LIN {X 0,Y 249.004,Z 223.47,A -85,B 0,C 180,E1 -19037.36,E2 -19037.36} C_VEL
LIN {X 0,Y 249.044,Z 223.457,A -85,B 0,C 180,E1 -19042.201,E2 -19042.201} C_VEL
LIN {X 0,Y 249.045,Z 223.461,A -85,B 0,C 180,E1 -19045.64,E2 -19045.64} C_VEL
LIN {X 0,Y 249.004,Z 223.467,A -85,B 0,C 180,E1 -19049.467,E2 -19049.467} C_VEL
LIN {X 0,Y 249.038,Z 223.46,A -85,B 0,C 180,E1 -19053.158,E2 -19053.158} C_VEL
LIN {X 0,Y 249.057,Z 223.459,A -85,B 0,C 180,E1 -19056.73,E2 -19056.73} C_VEL
LIN {X 0,Y 249.089,Z 223.455,A -85,B 0,C 180,E1 -19060.21,E2 -19060.21} C_VEL
LIN {X 0,Y 249.199,Z 223.439,A -85,B 0,C 180,E1 -19063.619,E2 -19063.619} C_VEL
LIN {X 0,Y 249.237,Z 223.426,A -85,B 0,C 180,E1 -19068.616,E2 -19068.616} C_VEL
LIN {X 0,Y 249.421,Z 223.401,A -85,B 0,C 180,E1 -19071.901,E2 -19071.901} C_VEL
LIN {X 0,Y 249.275,Z 223.429,A -85,B 0,C 180,E1 -19075.148,E2 -19075.148} C_VEL
LIN {X 0,Y 249.67,Z 223.386,A -85,B 0,C 180,E1 -19078.387,E2 -19078.387} C_VEL
LIN {X 0,Y 249.664,Z 223.384,A -85,B 0,C 180,E1 -19081.613,E2 -19081.613} C_VEL
LIN {X 0,Y 249.432,Z 223.406,A -85,B 0,C 180,E1 -19086.471,E2 -19086.471} C_VEL
LIN {X 0,Y 249.346,Z 223.417,A -85,B 0,C 180,E1 -19089.736,E2 -19089.736} C_VEL
LIN {X 0,Y 249.166,Z 223.447,A -85,B 0,C 180,E1 -19094.706,E2 -19094.706} C_VEL
LIN {X 0,Y 249.108,Z 223.454,A -85,B 0,C 180,E1 -19098.12,E2 -19098.12} C_VEL
LIN {X 0,Y 248.362,Z 223.545,A -85,B 0,C 180,E1 -19099.469,E2 -19099.469} C_VEL
LIN {X 0,Y 245.448,Z 223.906,A -85,B 0,C 180,E1 -19101.666,E2 -19101.666} C_VEL
LIN {X 0,Y 243.036,Z 224.209,A -85,B 0,C 180,E1 -19103.456,E2 -19103.456} C_VEL
LIN {X 0,Y 242.037,Z 224.335,A -85,B 0,C 180,E1 -19104.845,E2 -19104.845} C_VEL
LIN {X 0,Y 241.972,Z 224.344,A -85,B 0,C 180,E1 -19105.316,E2 -19105.316} C_VEL
LIN {X 0,Y 241.971,Z 224.343,A -85,B 0,C 180,E1 -19109.588,E2 -19109.588} C_VEL
LIN {X 0,Y 241.982,Z 224.344,A -85,B 0,C 180,E1 -19113.493,E2 -19113.493} C_VEL
LIN {X 0,Y 241.986,Z 224.345,A -85,B 0,C 180,E1 -19117.583,E2 -19117.583} C_VEL
LIN {X 0,Y 241.912,Z 224.352,A -85,B 0,C 180,E1 -19121.928,E2 -19121.928} C_VEL
LIN {X 0,Y 241.903,Z 224.351,A -85,B 0,C 180,E1 -19126.58,E2 -19126.58} C_VEL
LIN {X 0,Y 241.997,Z 224.342,A -85,B 0,C 180,E1 -19131.64,E2 -19131.64} C_VEL
LIN {X 0,Y 242.029,Z 224.408,A -85,B 0,C 180,E1 -19132.328,E2 -19132.328} C_VEL
LIN {X 0,Y 244.612,Z 236.152,A -85,B 0,C 180,E1 -19136.43,E2 -19136.43} C_VEL
LIN {X 0,Y 247.148,Z 248.776,A -85,B 0,C 180,E1 -19140.577,E2 -19140.577} C_VEL
LIN {X 0,Y 249.712,Z 271.884,A -85,B 0,C 180,E1 -19141.664,E2 -19141.664} C_VEL
LIN {X 0,Y 253.2,Z 306.04,A -85,B 0,C 180,E1 -19143.192,E2 -19143.192} C_VEL
LIN {X 0,Y 251.212,Z 359.282,A -85,B 0,C 180,E1 -19145.022,E2 -19145.022} C_VEL
LIN {X 0,Y 250.257,Z 372.001,A -85,B 0,C 180,E1 -19145.75,E2 -19145.75} C_VEL
LIN {X 0,Y 248.888,Z 385.038,A -85,B 0,C 180,E1 -19146.823,E2 -19146.823} C_VEL
LIN {X 0,Y 247.113,Z 398.148,A -85,B 0,C 180,E1 -19148.301,E2 -19148.301} C_VEL
LIN {X 0,Y 245.54,Z 409.14,A -85,B 0,C 180,E1 -19149.911,E2 -19149.911} C_VEL
LIN {X 0,Y 243.962,Z 419.427,A -85,B 0,C 180,E1 -19151.814,E2 -19151.814} C_VEL
LIN {X 0,Y 242.778,Z 427.354,A -85,B 0,C 180,E1 -19153.605,E2 -19153.605} C_VEL
LIN {X 0,Y 241.628,Z 436.389,A -85,B 0,C 180,E1 -19156.115,E2 -19156.115} C_VEL
LIN {X 0,Y 240.728,Z 443.544,A -85,B 0,C 180,E1 -19158.634,E2 -19158.634} C_VEL
LIN {X 0,Y 240.323,Z 450.068,A -85,B 0,C 180,E1 -19161.592,E2 -19161.592} C_VEL
LIN {X 0,Y 240.317,Z 453.94,A -85,B 0,C 180,E1 -19163.892,E2 -19163.892} C_VEL
LIN {X 0,Y 240.292,Z 457.328,A -85,B 0,C 180,E1 -19166.646,E2 -19166.646} C_VEL
LIN {X 0,Y 240.448,Z 458.797,A -85,B 0,C 180,E1 -19168.325,E2 -19168.325} C_VEL
LIN {X 0,Y 240.644,Z 459.779,A -85,B 0,C 180,E1 -19170,E2 -19170} C_VEL
LIN {X 0,Y 240.335,Z 460.292,A -85,B 0,C 180,E1 -19171.675,E2 -19171.675} C_VEL
LIN {X 0,Y 240.15,Z 460.406,A -85,B 0,C 180,E1 -19173.355,E2 -19173.355} C_VEL
LIN {X 0,Y 239.968,Z 460.015,A -85,B 0,C 180,E1 -19175.272,E2 -19175.272} C_VEL
LIN {X 0,Y 240.126,Z 458.23,A -85,B 0,C 180,E1 -19178.414,E2 -19178.414} C_VEL
LIN {X 0,Y 240.395,Z 456.694,A -85,B 0,C 180,E1 -19180.102,E2 -19180.102} C_VEL
LIN {X 0,Y 241.109,Z 453.576,A -85,B 0,C 180,E1 -19182.627,E2 -19182.627} C_VEL
LIN {X 0,Y 242.499,Z 449.461,A -85,B 0,C 180,E1 -19185.119,E2 -19185.119} C_VEL
LIN {X 0,Y 244.576,Z 443.266,A -85,B 0,C 180,E1 -19187.993,E2 -19187.993} C_VEL
LIN {X 0,Y 246.746,Z 436.536,A -85,B 0,C 180,E1 -19190.42,E2 -19190.42} C_VEL
LIN {X 0,Y 249.644,Z 428.244,A -85,B 0,C 180,E1 -19192.773,E2 -19192.773} C_VEL
LIN {X 0,Y 253.105,Z 418.103,A -85,B 0,C 180,E1 -19195.052,E2 -19195.052} C_VEL
LIN {X 0,Y 256.227,Z 407.616,A -85,B 0,C 180,E1 -19196.909,E2 -19196.909} C_VEL
LIN {X 0,Y 259.456,Z 395.965,A -85,B 0,C 180,E1 -19198.516,E2 -19198.516} C_VEL
LIN {X 0,Y 262.177,Z 384.572,A -85,B 0,C 180,E1 -19199.73,E2 -19199.73} C_VEL
LIN {X 0,Y 264.726,Z 371.887,A -85,B 0,C 180,E1 -19200.734,E2 -19200.734} C_VEL
LIN {X 0,Y 266.699,Z 358.144,A -85,B 0,C 180,E1 -19201.528,E2 -19201.528} C_VEL
LIN {X 0,Y 268.166,Z 340.024,A -85,B 0,C 180,E1 -19202.191,E2 -19202.191} C_VEL
LIN {X 0,Y 270.151,Z 309.712,A -85,B 0,C 180,E1 -19203.199,E2 -19203.199} C_VEL
LIN {X 0,Y 268.902,Z 293.084,A -85,B 0,C 180,E1 -19204.25,E2 -19204.25} C_VEL
LIN {X 0,Y 266.92,Z 276.84,A -85,B 0,C 180,E1 -19205.487,E2 -19205.487} C_VEL
LIN {X 0,Y 263.665,Z 268.777,A -85,B 0,C 180,E1 -19206.696,E2 -19206.696} C_VEL
LIN {X 0,Y 259.896,Z 260.954,A -85,B 0,C 180,E1 -19208.095,E2 -19208.095} C_VEL
LIN {X 0,Y 257.167,Z 255.727,A -85,B 0,C 180,E1 -19209.168,E2 -19209.168} C_VEL
LIN {X 0,Y 254.586,Z 251.104,A -85,B 0,C 180,E1 -19210.228,E2 -19210.228} C_VEL
LIN {X 0,Y 250.869,Z 244.957,A -85,B 0,C 180,E1 -19211.84,E2 -19211.84} C_VEL
LIN {X 0,Y 246.986,Z 238.614,A -85,B 0,C 180,E1 -19213.774,E2 -19213.774} C_VEL
LIN {X 0,Y 244.929,Z 232.476,A -85,B 0,C 180,E1 -19217.6,E2 -19217.6} C_VEL
LIN {X 0,Y 243.229,Z 227.568,A -85,B 0,C 180,E1 -19221.274,E2 -19221.274} C_VEL
LIN {X 0,Y 242.005,Z 224.336,A -85,B 0,C 180,E1 -19224.403,E2 -19224.403} C_VEL
LIN {X 0,Y 241.953,Z 224.342,A -85,B 0,C 180,E1 -19228.476,E2 -19228.476} C_VEL
LIN {X 0,Y 241.969,Z 224.343,A -85,B 0,C 180,E1 -19232.308,E2 -19232.308} C_VEL
LIN {X 0,Y 242.026,Z 224.331,A -85,B 0,C 180,E1 -19236.012,E2 -19236.012} C_VEL
LIN {X 0,Y 242.022,Z 224.33,A -85,B 0,C 180,E1 -19239.606,E2 -19239.606} C_VEL
LIN {X 0,Y 242.115,Z 224.321,A -85,B 0,C 180,E1 -19243.316,E2 -19243.316} C_VEL
LIN {X 0,Y 242.154,Z 224.318,A -85,B 0,C 180,E1 -19246.574,E2 -19246.574} C_VEL
LIN {X 0,Y 242.4,Z 224.286,A -85,B 0,C 180,E1 -19251.664,E2 -19251.664} C_VEL
LIN {X 0,Y 242.421,Z 224.433,A -85,B 0,C 180,E1 -19252.451,E2 -19252.451} C_VEL
LIN {X 0,Y 243.17,Z 226.719,A -85,B 0,C 180,E1 -19252.996,E2 -19252.996} C_VEL
LIN {X 0,Y 245.186,Z 229.149,A -85,B 0,C 180,E1 -19254.098,E2 -19254.098} C_VEL
LIN {X 0,Y 246.596,Z 230.283,A -85,B 0,C 180,E1 -19254.789,E2 -19254.789} C_VEL
LIN {X 0,Y 248.318,Z 233.194,A -85,B 0,C 180,E1 -19255.688,E2 -19255.688} C_VEL
LIN {X 0,Y 250.915,Z 235.599,A -85,B 0,C 180,E1 -19256.82,E2 -19256.82} C_VEL
LIN {X 0,Y 253.281,Z 239.028,A -85,B 0,C 180,E1 -19257.877,E2 -19257.877} C_VEL
LIN {X 0,Y 254.718,Z 240.902,A -85,B 0,C 180,E1 -19258.464,E2 -19258.464} C_VEL
LIN {X 0,Y 257.831,Z 245.506,A -85,B 0,C 180,E1 -19259.698,E2 -19259.698} C_VEL
LIN {X 0,Y 265.688,Z 258.053,A -85,B 0,C 180,E1 -19262.526,E2 -19262.526} C_VEL
LIN {X 0,Y 270.454,Z 266.96,A -85,B 0,C 180,E1 -19264.103,E2 -19264.103} C_VEL
LIN {X 0,Y 272.41,Z 270.959,A -85,B 0,C 180,E1 -19264.719,E2 -19264.719} C_VEL
LIN {X 0,Y 268.634,Z 326.119,A -85,B 0,C 180,E1 -19266.582,E2 -19266.582} C_VEL
LIN {X 0,Y 267.326,Z 338.992,A -85,B 0,C 180,E1 -19267.297,E2 -19267.297} C_VEL
LIN {X 0,Y 265.555,Z 351.406,A -85,B 0,C 180,E1 -19268.274,E2 -19268.274} C_VEL
LIN {X 0,Y 263.204,Z 363.778,A -85,B 0,C 180,E1 -19269.568,E2 -19269.568} C_VEL
LIN {X 0,Y 260.667,Z 374.697,A -85,B 0,C 180,E1 -19271.046,E2 -19271.046} C_VEL
LIN {X 0,Y 257.859,Z 384.956,A -85,B 0,C 180,E1 -19272.794,E2 -19272.794} C_VEL
LIN {X 0,Y 254.955,Z 394.175,A -85,B 0,C 180,E1 -19274.783,E2 -19274.783} C_VEL
LIN {X 0,Y 252.106,Z 402.348,A -85,B 0,C 180,E1 -19276.998,E2 -19276.998} C_VEL
LIN {X 0,Y 249.515,Z 409.181,A -85,B 0,C 180,E1 -19279.327,E2 -19279.327} C_VEL
LIN {X 0,Y 247.225,Z 414.655,A -85,B 0,C 180,E1 -19281.688,E2 -19281.688} C_VEL
LIN {X 0,Y 244.992,Z 419.645,A -85,B 0,C 180,E1 -19284.579,E2 -19284.579} C_VEL
LIN {X 0,Y 243.177,Z 423.206,A -85,B 0,C 180,E1 -19287.543,E2 -19287.543} C_VEL
LIN {X 0,Y 242.202,Z 424.804,A -85,B 0,C 180,E1 -19289.557,E2 -19289.557} C_VEL
LIN {X 0,Y 241.18,Z 425.997,A -85,B 0,C 180,E1 -19292.322,E2 -19292.322} C_VEL
LIN {X 0,Y 240.526,Z 426.078,A -85,B 0,C 180,E1 -19295.102,E2 -19295.102} C_VEL
LIN {X 0,Y 240.229,Z 425.025,A -85,B 0,C 180,E1 -19297.906,E2 -19297.906} C_VEL
LIN {X 0,Y 240.205,Z 423.052,A -85,B 0,C 180,E1 -19300.473,E2 -19300.473} C_VEL
LIN {X 0,Y 240.581,Z 419.994,A -85,B 0,C 180,E1 -19303.088,E2 -19303.088} C_VEL
LIN {X 0,Y 241.163,Z 415.077,A -85,B 0,C 180,E1 -19306.098,E2 -19306.098} C_VEL
LIN {X 0,Y 241.859,Z 409.983,A -85,B 0,C 180,E1 -19308.464,E2 -19308.464} C_VEL
LIN {X 0,Y 242.782,Z 403.678,A -85,B 0,C 180,E1 -19310.816,E2 -19310.816} C_VEL
LIN {X 0,Y 244.097,Z 395.086,A -85,B 0,C 180,E1 -19313.375,E2 -19313.375} C_VEL
LIN {X 0,Y 245.483,Z 385.904,A -85,B 0,C 180,E1 -19315.575,E2 -19315.575} C_VEL
LIN {X 0,Y 246.977,Z 375.589,A -85,B 0,C 180,E1 -19317.553,E2 -19317.553} C_VEL
LIN {X 0,Y 248.499,Z 363.511,A -85,B 0,C 180,E1 -19319.398,E2 -19319.398} C_VEL
LIN {X 0,Y 249.898,Z 351.267,A -85,B 0,C 180,E1 -19320.836,E2 -19320.836} C_VEL
LIN {X 0,Y 251.035,Z 338.511,A -85,B 0,C 180,E1 -19321.971,E2 -19321.971} C_VEL
LIN {X 0,Y 251.729,Z 325.929,A -85,B 0,C 180,E1 -19322.781,E2 -19322.781} C_VEL
LIN {X 0,Y 252.39,Z 309.148,A -85,B 0,C 180,E1 -19323.438,E2 -19323.438} C_VEL
LIN {X 0,Y 254.486,Z 255.593,A -85,B 0,C 180,E1 -19325.202,E2 -19325.202} C_VEL
LIN {X 0,Y 244.932,Z 231.694,A -85,B 0,C 180,E1 -19326.909,E2 -19326.909} C_VEL
LIN {X 0,Y 242.099,Z 224.79,A -85,B 0,C 180,E1 -19327.436,E2 -19327.436} C_VEL
LIN {X 0,Y 242.005,Z 224.341,A -85,B 0,C 180,E1 -19327.483,E2 -19327.483} C_VEL
LIN {X 0,Y 242.05,Z 224.334,A -85,B 0,C 180,E1 -19331.375,E2 -19331.375} C_VEL
LIN {X 0,Y 242.14,Z 224.324,A -85,B 0,C 180,E1 -19334.858,E2 -19334.858} C_VEL
LIN {X 0,Y 242.343,Z 224.299,A -85,B 0,C 180,E1 -19340.405,E2 -19340.405} C_VEL
LIN {X 0,Y 242.401,Z 224.289,A -85,B 0,C 180,E1 -19343.341,E2 -19343.341} C_VEL
LIN {X 0,Y 242.634,Z 224.262,A -85,B 0,C 180,E1 -19348.341,E2 -19348.341} C_VEL
LIN {X 0,Y 242.632,Z 224.259,A -85,B 0,C 180,E1 -19351.66,E2 -19351.66} C_VEL
LIN {X 0,Y 242.408,Z 224.289,A -85,B 0,C 180,E1 -19356.66,E2 -19356.66} C_VEL
LIN {X 0,Y 242.269,Z 224.307,A -85,B 0,C 180,E1 -19360.024,E2 -19360.024} C_VEL
LIN {X 0,Y 242.169,Z 224.317,A -85,B 0,C 180,E1 -19365.141,E2 -19365.141} C_VEL
LIN {X 0,Y 242.074,Z 224.327,A -85,B 0,C 180,E1 -19368.625,E2 -19368.625} C_VEL
LIN {X 0,Y 242.007,Z 224.332,A -85,B 0,C 180,E1 -19372.181,E2 -19372.181} C_VEL
LIN {X 0,Y 242.034,Z 224.335,A -85,B 0,C 180,E1 -19375.821,E2 -19375.821} C_VEL
LIN {X 0,Y 241.971,Z 224.345,A -85,B 0,C 180,E1 -19379.589,E2 -19379.589} C_VEL
LIN {X 0,Y 241.981,Z 224.34,A -85,B 0,C 180,E1 -19383.493,E2 -19383.493} C_VEL
LIN {X 0,Y 241.985,Z 224.327,A -85,B 0,C 180,E1 -19387.583,E2 -19387.583} C_VEL
LIN {X 0,Y 241.929,Z 224.344,A -85,B 0,C 180,E1 -19391.925,E2 -19391.925} C_VEL
LIN {X 0,Y 241.922,Z 224.348,A -85,B 0,C 180,E1 -19396.575,E2 -19396.575} C_VEL
LIN {X 0,Y 241.995,Z 224.337,A -85,B 0,C 180,E1 -19401.641,E2 -19401.641} C_VEL
LIN {X 0,Y 241.989,Z 224.336,A -85,B 0,C 180,E1 -19404.489,E2 -19404.489} C_VEL
LIN {X 0,Y 241.955,Z 224.344,A -85,B 0,C 180,E1 -19408.477,E2 -19408.477} C_VEL
LIN {X 0,Y 241.97,Z 224.34,A -85,B 0,C 180,E1 -19412.308,E2 -19412.308} C_VEL
LIN {X 0,Y 242.027,Z 224.331,A -85,B 0,C 180,E1 -19416.013,E2 -19416.013} C_VEL
LIN {X 0,Y 242.024,Z 224.335,A -85,B 0,C 180,E1 -19419.607,E2 -19419.607} C_VEL
LIN {X 0,Y 242.13,Z 224.32,A -85,B 0,C 180,E1 -19423.307,E2 -19423.307} C_VEL
LIN {X 0,Y 242.171,Z 224.308,A -85,B 0,C 180,E1 -19428.279,E2 -19428.279} C_VEL
LIN {X 0,Y 242.375,Z 224.277,A -85,B 0,C 180,E1 -19431.664,E2 -19431.664} C_VEL
LIN {X 0,Y 242.236,Z 224.306,A -85,B 0,C 180,E1 -19435.007,E2 -19435.007} C_VEL
LIN {X 0,Y 242.63,Z 224.262,A -85,B 0,C 180,E1 -19438.34,E2 -19438.34} C_VEL
LIN {X 0,Y 242.623,Z 224.261,A -85,B 0,C 180,E1 -19441.66,E2 -19441.66} C_VEL
LIN {X 0,Y 242.404,Z 224.279,A -85,B 0,C 180,E1 -19446.66,E2 -19446.66} C_VEL
LIN {X 0,Y 242.269,Z 224.3,A -85,B 0,C 180,E1 -19450.024,E2 -19450.024} C_VEL
LIN {X 0,Y 242.129,Z 224.324,A -85,B 0,C 180,E1 -19455.143,E2 -19455.143} C_VEL
LIN {X 0,Y 242.049,Z 224.331,A -85,B 0,C 180,E1 -19458.626,E2 -19458.626} C_VEL
LIN {X 0,Y 241.991,Z 224.339,A -85,B 0,C 180,E1 -19462.182,E2 -19462.182} C_VEL
LIN {X 0,Y 241.972,Z 224.344,A -85,B 0,C 180,E1 -19465.316,E2 -19465.316} C_VEL
LIN {X 0,Y 241.353,Z 224.425,A -85,B 0,C 180,E1 -19466.705,E2 -19466.705} C_VEL
LIN {X 0,Y 238.537,Z 224.775,A -85,B 0,C 180,E1 -19468.972,E2 -19468.972} C_VEL
LIN {X 0,Y 236.106,Z 225.073,A -85,B 0,C 180,E1 -19470.819,E2 -19470.819} C_VEL
LIN {X 0,Y 235.045,Z 225.205,A -85,B 0,C 180,E1 -19472.252,E2 -19472.252} C_VEL
LIN {X 0,Y 234.95,Z 225.216,A -85,B 0,C 180,E1 -19472.738,E2 -19472.738} C_VEL
LIN {X 0,Y 234.918,Z 225.221,A -85,B 0,C 180,E1 -19476.751,E2 -19476.751} C_VEL
LIN {X 0,Y 234.914,Z 225.224,A -85,B 0,C 180,E1 -19478.935,E2 -19478.935} C_VEL
LIN {X 0,Y 234.855,Z 225.233,A -85,B 0,C 180,E1 -19483.494,E2 -19483.494} C_VEL
LIN {X 0,Y 234.856,Z 225.229,A -85,B 0,C 180,E1 -19486.506,E2 -19486.506} C_VEL
LIN {X 0,Y 234.972,Z 225.217,A -85,B 0,C 180,E1 -19491.774,E2 -19491.774} C_VEL
LIN {X 0,Y 236.986,Z 234.459,A -85,B 0,C 180,E1 -19495.188,E2 -19495.188} C_VEL
LIN {X 0,Y 239.364,Z 245.731,A -85,B 0,C 180,E1 -19499.082,E2 -19499.082} C_VEL
LIN {X 0,Y 239.85,Z 248.256,A -85,B 0,C 180,E1 -19499.905,E2 -19499.905} C_VEL
LIN {X 0,Y 241.048,Z 253.117,A -85,B 0,C 180,E1 -19500.204,E2 -19500.204} C_VEL
LIN {X 0,Y 246.464,Z 306.984,A -85,B 0,C 180,E1 -19502.71,E2 -19502.71} C_VEL
LIN {X 0,Y 244.423,Z 358.04,A -85,B 0,C 180,E1 -19504.506,E2 -19504.506} C_VEL
LIN {X 0,Y 243.525,Z 370.993,A -85,B 0,C 180,E1 -19505.262,E2 -19505.262} C_VEL
LIN {X 0,Y 242.077,Z 384.148,A -85,B 0,C 180,E1 -19506.358,E2 -19506.358} C_VEL
LIN {X 0,Y 240.52,Z 395.755,A -85,B 0,C 180,E1 -19507.674,E2 -19507.674} C_VEL
LIN {X 0,Y 238.876,Z 407.102,A -85,B 0,C 180,E1 -19509.325,E2 -19509.325} C_VEL
LIN {X 0,Y 237.422,Z 416.33,A -85,B 0,C 180,E1 -19510.997,E2 -19510.997} C_VEL
LIN {X 0,Y 235.854,Z 425.804,A -85,B 0,C 180,E1 -19513.11,E2 -19513.11} C_VEL
LIN {X 0,Y 234.679,Z 435.015,A -85,B 0,C 180,E1 -19515.696,E2 -19515.696} C_VEL
LIN {X 0,Y 233.729,Z 442.37,A -85,B 0,C 180,E1 -19518.289,E2 -19518.289} C_VEL
LIN {X 0,Y 233.34,Z 447.316,A -85,B 0,C 180,E1 -19520.464,E2 -19520.464} C_VEL
LIN {X 0,Y 233.202,Z 452.07,A -85,B 0,C 180,E1 -19523.076,E2 -19523.076} C_VEL
LIN {X 0,Y 233.272,Z 454.555,A -85,B 0,C 180,E1 -19524.814,E2 -19524.814} C_VEL
LIN {X 0,Y 233.225,Z 456.519,A -85,B 0,C 180,E1 -19526.544,E2 -19526.544} C_VEL
LIN {X 0,Y 233.365,Z 458.051,A -85,B 0,C 180,E1 -19528.274,E2 -19528.274} C_VEL
LIN {X 0,Y 233.587,Z 459.122,A -85,B 0,C 180,E1 -19530,E2 -19530} C_VEL
LIN {X 0,Y 233.249,Z 459.681,A -85,B 0,C 180,E1 -19531.726,E2 -19531.726} C_VEL
LIN {X 0,Y 233.071,Z 459.842,A -85,B 0,C 180,E1 -19533.457,E2 -19533.457} C_VEL
LIN {X 0,Y 232.897,Z 459.588,A -85,B 0,C 180,E1 -19535.237,E2 -19535.237} C_VEL
LIN {X 0,Y 232.899,Z 458.941,A -85,B 0,C 180,E1 -19536.932,E2 -19536.932} C_VEL
LIN {X 0,Y 233.373,Z 456.383,A -85,B 0,C 180,E1 -19540.409,E2 -19540.409} C_VEL
LIN {X 0,Y 234.161,Z 453.382,A -85,B 0,C 180,E1 -19543.008,E2 -19543.008} C_VEL
LIN {X 0,Y 235.638,Z 449.379,A -85,B 0,C 180,E1 -19545.57,E2 -19545.57} C_VEL
LIN {X 0,Y 237.455,Z 444.269,A -85,B 0,C 180,E1 -19548.105,E2 -19548.105} C_VEL
LIN {X 0,Y 239.664,Z 437.95,A -85,B 0,C 180,E1 -19550.603,E2 -19550.603} C_VEL
LIN {X 0,Y 242.605,Z 430.206,A -85,B 0,C 180,E1 -19553.021,E2 -19553.021} C_VEL
LIN {X 0,Y 245.465,Z 422.389,A -85,B 0,C 180,E1 -19554.98,E2 -19554.98} C_VEL
LIN {X 0,Y 248.945,Z 411.937,A -85,B 0,C 180,E1 -19557.079,E2 -19557.079} C_VEL
LIN {X 0,Y 252.189,Z 401.412,A -85,B 0,C 180,E1 -19558.732,E2 -19558.732} C_VEL
LIN {X 0,Y 255.304,Z 389.924,A -85,B 0,C 180,E1 -19560.157,E2 -19560.157} C_VEL
LIN {X 0,Y 258.063,Z 378.066,A -85,B 0,C 180,E1 -19561.274,E2 -19561.274} C_VEL
LIN {X 0,Y 260.595,Z 364.125,A -85,B 0,C 180,E1 -19562.241,E2 -19562.241} C_VEL
LIN {X 0,Y 262.232,Z 350.287,A -85,B 0,C 180,E1 -19562.895,E2 -19562.895} C_VEL
LIN {X 0,Y 265.041,Z 310.297,A -85,B 0,C 180,E1 -19564.251,E2 -19564.251} C_VEL
LIN {X 0,Y 263.895,Z 294.774,A -85,B 0,C 180,E1 -19565.275,E2 -19565.275} C_VEL
LIN {X 0,Y 262.209,Z 279.646,A -85,B 0,C 180,E1 -19566.477,E2 -19566.477} C_VEL
LIN {X 0,Y 257.444,Z 268.533,A -85,B 0,C 180,E1 -19568.335,E2 -19568.335} C_VEL
LIN {X 0,Y 253.621,Z 260.876,A -85,B 0,C 180,E1 -19569.925,E2 -19569.925} C_VEL
LIN {X 0,Y 251.077,Z 256.261,A -85,B 0,C 180,E1 -19571.019,E2 -19571.019} C_VEL
LIN {X 0,Y 247.526,Z 250.181,A -85,B 0,C 180,E1 -19572.681,E2 -19572.681} C_VEL
LIN {X 0,Y 243.577,Z 243.84,A -85,B 0,C 180,E1 -19574.706,E2 -19574.706} C_VEL
LIN {X 0,Y 239.557,Z 237.626,A -85,B 0,C 180,E1 -19577.067,E2 -19577.067} C_VEL
LIN {X 0,Y 239.211,Z 236.801,A -85,B 0,C 180,E1 -19577.488,E2 -19577.488} C_VEL
LIN {X 0,Y 237.935,Z 233.255,A -85,B 0,C 180,E1 -19580.172,E2 -19580.172} C_VEL
LIN {X 0,Y 237.409,Z 231.555,A -85,B 0,C 180,E1 -19581.562,E2 -19581.562} C_VEL
LIN {X 0,Y 235.745,Z 227.774,A -85,B 0,C 180,E1 -19585.498,E2 -19585.498} C_VEL
LIN {X 0,Y 234.888,Z 225.226,A -85,B 0,C 180,E1 -19588.927,E2 -19588.927} C_VEL
LIN {X 0,Y 234.968,Z 225.209,A -85,B 0,C 180,E1 -19593.806,E2 -19593.806} C_VEL
LIN {X 0,Y 234.99,Z 225.208,A -85,B 0,C 180,E1 -19598.968,E2 -19598.968} C_VEL
LIN {X 0,Y 235.056,Z 225.199,A -85,B 0,C 180,E1 -19603.092,E2 -19603.092} C_VEL
LIN {X 0,Y 235.111,Z 225.192,A -85,B 0,C 180,E1 -19607.922,E2 -19607.922} C_VEL
LIN {X 0,Y 235.173,Z 225.364,A -85,B 0,C 180,E1 -19608.471,E2 -19608.471} C_VEL
LIN {X 0,Y 235.883,Z 227.535,A -85,B 0,C 180,E1 -19609.175,E2 -19609.175} C_VEL
LIN {X 0,Y 237.812,Z 229.766,A -85,B 0,C 180,E1 -19610.554,E2 -19610.554} C_VEL
LIN {X 0,Y 239.977,Z 231.128,A -85,B 0,C 180,E1 -19611.844,E2 -19611.844} C_VEL
LIN {X 0,Y 241.504,Z 234.067,A -85,B 0,C 180,E1 -19612.853,E2 -19612.853} C_VEL
LIN {X 0,Y 244.057,Z 236.636,A -85,B 0,C 180,E1 -19614.215,E2 -19614.215} C_VEL
LIN {X 0,Y 246.175,Z 239.881,A -85,B 0,C 180,E1 -19615.353,E2 -19615.353} C_VEL
LIN {X 0,Y 248.301,Z 242.029,A -85,B 0,C 180,E1 -19616.317,E2 -19616.317} C_VEL
LIN {X 0,Y 251.891,Z 247.07,A -85,B 0,C 180,E1 -19617.942,E2 -19617.942} C_VEL
LIN {X 0,Y 255.949,Z 253.269,A -85,B 0,C 180,E1 -19619.606,E2 -19619.606} C_VEL
LIN {X 0,Y 262.708,Z 264.58,A -85,B 0,C 180,E1 -19622.126,E2 -19622.126} C_VEL
LIN {X 0,Y 267.253,Z 273.702,A -85,B 0,C 180,E1 -19623.724,E2 -19623.724} C_VEL
LIN {X 0,Y 263.345,Z 327.819,A -85,B 0,C 180,E1 -19625.592,E2 -19625.592} C_VEL
LIN {X 0,Y 261.967,Z 340.677,A -85,B 0,C 180,E1 -19626.344,E2 -19626.344} C_VEL
LIN {X 0,Y 259.996,Z 353.314,A -85,B 0,C 180,E1 -19627.377,E2 -19627.377} C_VEL
LIN {X 0,Y 257.339,Z 366.137,A -85,B 0,C 180,E1 -19628.796,E2 -19628.796} C_VEL
LIN {X 0,Y 254.63,Z 376.895,A -85,B 0,C 180,E1 -19630.335,E2 -19630.335} C_VEL
LIN {X 0,Y 251.616,Z 386.962,A -85,B 0,C 180,E1 -19632.151,E2 -19632.151} C_VEL
LIN {X 0,Y 248.365,Z 396.576,A -85,B 0,C 180,E1 -19634.335,E2 -19634.335} C_VEL
LIN {X 0,Y 245.362,Z 404.543,A -85,B 0,C 180,E1 -19636.645,E2 -19636.645} C_VEL
LIN {X 0,Y 242.676,Z 410.983,A -85,B 0,C 180,E1 -19639.014,E2 -19639.014} C_VEL
LIN {X 0,Y 240.198,Z 416.421,A -85,B 0,C 180,E1 -19641.581,E2 -19641.581} C_VEL
LIN {X 0,Y 238.003,Z 420.922,A -85,B 0,C 180,E1 -19644.419,E2 -19644.419} C_VEL
LIN {X 0,Y 236.433,Z 423.731,A -85,B 0,C 180,E1 -19646.906,E2 -19646.906} C_VEL
LIN {X 0,Y 234.991,Z 425.851,A -85,B 0,C 180,E1 -19649.852,E2 -19649.852} C_VEL
LIN {X 0,Y 233.985,Z 426.73,A -85,B 0,C 180,E1 -19652.754,E2 -19652.754} C_VEL
LIN {X 0,Y 233.369,Z 426.465,A -85,B 0,C 180,E1 -19655.599,E2 -19655.599} C_VEL
LIN {X 0,Y 233.107,Z 425.142,A -85,B 0,C 180,E1 -19658.383,E2 -19658.383} C_VEL
LIN {X 0,Y 233.211,Z 422.328,A -85,B 0,C 180,E1 -19661.528,E2 -19661.528} C_VEL
LIN {X 0,Y 233.59,Z 419.419,A -85,B 0,C 180,E1 -19663.788,E2 -19663.788} C_VEL
LIN {X 0,Y 234.145,Z 415.112,A -85,B 0,C 180,E1 -19666.342,E2 -19666.342} C_VEL
LIN {X 0,Y 235.022,Z 408.743,A -85,B 0,C 180,E1 -19669.243,E2 -19669.243} C_VEL
LIN {X 0,Y 236.105,Z 401.648,A -85,B 0,C 180,E1 -19671.791,E2 -19671.791} C_VEL
LIN {X 0,Y 237.472,Z 393.305,A -85,B 0,C 180,E1 -19674.187,E2 -19674.187} C_VEL
LIN {X 0,Y 238.938,Z 383.199,A -85,B 0,C 180,E1 -19676.518,E2 -19676.518} C_VEL
LIN {X 0,Y 240.302,Z 373.997,A -85,B 0,C 180,E1 -19678.235,E2 -19678.235} C_VEL
LIN {X 0,Y 241.706,Z 363.056,A -85,B 0,C 180,E1 -19679.896,E2 -19679.896} C_VEL
LIN {X 0,Y 243.179,Z 350.224,A -85,B 0,C 180,E1 -19681.402,E2 -19681.402} C_VEL
LIN {X 0,Y 244.284,Z 338.134,A -85,B 0,C 180,E1 -19682.477,E2 -19682.477} C_VEL
LIN {X 0,Y 244.978,Z 325.026,A -85,B 0,C 180,E1 -19683.309,E2 -19683.309} C_VEL
LIN {X 0,Y 245.801,Z 304.619,A -85,B 0,C 180,E1 -19684.085,E2 -19684.085} C_VEL
LIN {X 0,Y 247.705,Z 256.997,A -85,B 0,C 180,E1 -19685.708,E2 -19685.708} C_VEL
LIN {X 0,Y 237.805,Z 232.408,A -85,B 0,C 180,E1 -19687.541,E2 -19687.541} C_VEL
LIN {X 0,Y 235.054,Z 225.62,A -85,B 0,C 180,E1 -19688.075,E2 -19688.075} C_VEL
LIN {X 0,Y 234.989,Z 225.214,A -85,B 0,C 180,E1 -19688.136,E2 -19688.136} C_VEL
LIN {X 0,Y 235.064,Z 225.205,A -85,B 0,C 180,E1 -19693.086,E2 -19693.086} C_VEL
LIN {X 0,Y 235.101,Z 225.199,A -85,B 0,C 180,E1 -19697.922,E2 -19697.922} C_VEL
LIN {X 0,Y 235.313,Z 225.173,A -85,B 0,C 180,E1 -19701.412,E2 -19701.412} C_VEL
LIN {X 0,Y 235.352,Z 225.168,A -85,B 0,C 180,E1 -19703.14,E2 -19703.14} C_VEL
LIN {X 0,Y 235.594,Z 225.138,A -85,B 0,C 180,E1 -19708.291,E2 -19708.291} C_VEL
LIN {X 0,Y 235.591,Z 225.136,A -85,B 0,C 180,E1 -19711.71,E2 -19711.71} C_VEL
LIN {X 0,Y 235.36,Z 225.166,A -85,B 0,C 180,E1 -19716.86,E2 -19716.86} C_VEL
LIN {X 0,Y 235.216,Z 225.187,A -85,B 0,C 180,E1 -19720.328,E2 -19720.328} C_VEL
LIN {X 0,Y 235.116,Z 225.197,A -85,B 0,C 180,E1 -19725.607,E2 -19725.607} C_VEL
LIN {X 0,Y 235.009,Z 225.206,A -85,B 0,C 180,E1 -19729.206,E2 -19729.206} C_VEL
LIN {X 0,Y 234.949,Z 225.209,A -85,B 0,C 180,E1 -19732.885,E2 -19732.885} C_VEL
LIN {X 0,Y 234.947,Z 225.216,A -85,B 0,C 180,E1 -19736.661,E2 -19736.661} C_VEL
LIN {X 0,Y 234.901,Z 225.222,A -85,B 0,C 180,E1 -19740.573,E2 -19740.573} C_VEL
LIN {X 0,Y 234.927,Z 225.212,A -85,B 0,C 180,E1 -19744.639,E2 -19744.639} C_VEL
LIN {X 0,Y 234.913,Z 225.205,A -85,B 0,C 180,E1 -19748.936,E2 -19748.936} C_VEL
LIN {X 0,Y 234.878,Z 225.224,A -85,B 0,C 180,E1 -19753.489,E2 -19753.489} C_VEL
LIN {X 0,Y 234.875,Z 225.225,A -85,B 0,C 180,E1 -19756.511,E2 -19756.511} C_VEL
LIN {X 0,Y 234.919,Z 225.221,A -85,B 0,C 180,E1 -19761.079,E2 -19761.079} C_VEL
LIN {X 0,Y 234.932,Z 225.22,A -85,B 0,C 180,E1 -19765.362,E2 -19765.362} C_VEL
LIN {X 0,Y 234.901,Z 225.224,A -85,B 0,C 180,E1 -19769.428,E2 -19769.428} C_VEL
LIN {X 0,Y 234.971,Z 225.209,A -85,B 0,C 180,E1 -19773.807,E2 -19773.807} C_VEL
LIN {X 0,Y 234.993,Z 225.214,A -85,B 0,C 180,E1 -19778.968,E2 -19778.968} C_VEL
LIN {X 0,Y 235.066,Z 225.201,A -85,B 0,C 180,E1 -19783.086,E2 -19783.086} C_VEL
LIN {X 0,Y 235.103,Z 225.186,A -85,B 0,C 180,E1 -19787.922,E2 -19787.922} C_VEL
LIN {X 0,Y 235.314,Z 225.155,A -85,B 0,C 180,E1 -19791.412,E2 -19791.412} C_VEL
LIN {X 0,Y 235.352,Z 225.158,A -85,B 0,C 180,E1 -19793.14,E2 -19793.14} C_VEL
LIN {X 0,Y 235.59,Z 225.139,A -85,B 0,C 180,E1 -19798.291,E2 -19798.291} C_VEL
LIN {X 0,Y 235.582,Z 225.138,A -85,B 0,C 180,E1 -19801.71,E2 -19801.71} C_VEL
LIN {X 0,Y 235.356,Z 225.155,A -85,B 0,C 180,E1 -19806.86,E2 -19806.86} C_VEL
LIN {X 0,Y 235.214,Z 225.181,A -85,B 0,C 180,E1 -19810.328,E2 -19810.328} C_VEL
LIN {X 0,Y 235.077,Z 225.204,A -85,B 0,C 180,E1 -19815.609,E2 -19815.609} C_VEL
LIN {X 0,Y 234.99,Z 225.21,A -85,B 0,C 180,E1 -19819.207,E2 -19819.207} C_VEL
LIN {X 0,Y 234.928,Z 225.217,A -85,B 0,C 180,E1 -19822.886,E2 -19822.886} C_VEL
LIN {X 0,Y 234.929,Z 225.221,A -85,B 0,C 180,E1 -19826.663,E2 -19826.663} C_VEL
LIN {X 0,Y 234.901,Z 225.218,A -85,B 0,C 180,E1 -19830.572,E2 -19830.572} C_VEL
LIN {X 0,Y 234.95,Z 225.216,A -85,B 0,C 180,E1 -19832.738,E2 -19832.738} C_VEL
LIN {X 0,Y 234.268,Z 225.306,A -85,B 0,C 180,E1 -19834.169,E2 -19834.169} C_VEL
LIN {X 0,Y 231.433,Z 225.667,A -85,B 0,C 180,E1 -19836.503,E2 -19836.503} C_VEL
LIN {X 0,Y 228.17,Z 226.07,A -85,B 0,C 180,E1 -19839.384,E2 -19839.384} C_VEL
LIN {X 0,Y 227.805,Z 226.109,A -85,B 0,C 180,E1 -19840.382,E2 -19840.382} C_VEL
LIN {X 0,Y 227.812,Z 226.109,A -85,B 0,C 180,E1 -19845.199,E2 -19845.199} C_VEL
LIN {X 0,Y 227.803,Z 226.11,A -85,B 0,C 180,E1 -19849.618,E2 -19849.618} C_VEL
LIN {X 0,Y 227.906,Z 226.166,A -85,B 0,C 180,E1 -19851.39,E2 -19851.39} C_VEL
LIN {X 0,Y 230.109,Z 236.131,A -85,B 0,C 180,E1 -19855.109,E2 -19855.109} C_VEL
LIN {X 0,Y 232.504,Z 247.603,A -85,B 0,C 180,E1 -19859.177,E2 -19859.177} C_VEL
LIN {X 0,Y 234.498,Z 254.636,A -85,B 0,C 180,E1 -19859.662,E2 -19859.662} C_VEL
LIN {X 0,Y 239.718,Z 307.336,A -85,B 0,C 180,E1 -19862.201,E2 -19862.201} C_VEL
LIN {X 0,Y 237.643,Z 357.471,A -85,B 0,C 180,E1 -19864.019,E2 -19864.019} C_VEL
LIN {X 0,Y 236.712,Z 370.423,A -85,B 0,C 180,E1 -19864.794,E2 -19864.794} C_VEL
LIN {X 0,Y 235.307,Z 383.081,A -85,B 0,C 180,E1 -19865.869,E2 -19865.869} C_VEL
LIN {X 0,Y 233.696,Z 394.813,A -85,B 0,C 180,E1 -19867.219,E2 -19867.219} C_VEL
LIN {X 0,Y 231.999,Z 406.234,A -85,B 0,C 180,E1 -19868.916,E2 -19868.916} C_VEL
LIN {X 0,Y 230.383,Z 416.251,A -85,B 0,C 180,E1 -19870.781,E2 -19870.781} C_VEL
LIN {X 0,Y 228.777,Z 425.901,A -85,B 0,C 180,E1 -19873.031,E2 -19873.031} C_VEL
LIN {X 0,Y 227.574,Z 435.008,A -85,B 0,C 180,E1 -19875.696,E2 -19875.696} C_VEL
LIN {X 0,Y 226.633,Z 442.245,A -85,B 0,C 180,E1 -19878.371,E2 -19878.371} C_VEL
LIN {X 0,Y 226.214,Z 447.984,A -85,B 0,C 180,E1 -19881.063,E2 -19881.063} C_VEL
LIN {X 0,Y 226.197,Z 452.582,A -85,B 0,C 180,E1 -19883.853,E2 -19883.853} C_VEL
LIN {X 0,Y 226.159,Z 455.71,A -85,B 0,C 180,E1 -19886.436,E2 -19886.436} C_VEL
LIN {X 0,Y 226.283,Z 457.292,A -85,B 0,C 180,E1 -19888.22,E2 -19888.22} C_VEL
LIN {X 0,Y 226.53,Z 458.446,A -85,B 0,C 180,E1 -19890,E2 -19890} C_VEL
LIN {X 0,Y 226.163,Z 459.069,A -85,B 0,C 180,E1 -19891.78,E2 -19891.78} C_VEL
LIN {X 0,Y 225.993,Z 459.277,A -85,B 0,C 180,E1 -19893.565,E2 -19893.565} C_VEL
LIN {X 0,Y 225.819,Z 458.497,A -85,B 0,C 180,E1 -19897.151,E2 -19897.151} C_VEL
LIN {X 0,Y 226.004,Z 457.502,A -85,B 0,C 180,E1 -19898.944,E2 -19898.944} C_VEL
LIN {X 0,Y 226.815,Z 454.249,A -85,B 0,C 180,E1 -19902.527,E2 -19902.527} C_VEL
LIN {X 0,Y 228.192,Z 450.699,A -85,B 0,C 180,E1 -19905.176,E2 -19905.176} C_VEL
LIN {X 0,Y 229.967,Z 446.126,A -85,B 0,C 180,E1 -19907.794,E2 -19907.794} C_VEL
LIN {X 0,Y 232.586,Z 439.345,A -85,B 0,C 180,E1 -19910.795,E2 -19910.795} C_VEL
LIN {X 0,Y 235.534,Z 432.024,A -85,B 0,C 180,E1 -19913.288,E2 -19913.288} C_VEL
LIN {X 0,Y 239.095,Z 422.994,A -85,B 0,C 180,E1 -19915.693,E2 -19915.693} C_VEL
LIN {X 0,Y 242.709,Z 412.927,A -85,B 0,C 180,E1 -19917.834,E2 -19917.834} C_VEL
LIN {X 0,Y 246.072,Z 402.815,A -85,B 0,C 180,E1 -19919.516,E2 -19919.516} C_VEL
LIN {X 0,Y 249.697,Z 390.261,A -85,B 0,C 180,E1 -19921.143,E2 -19921.143} C_VEL
LIN {X 0,Y 252.564,Z 378.739,A -85,B 0,C 180,E1 -19922.27,E2 -19922.27} C_VEL
LIN {X 0,Y 255.207,Z 365.183,A -85,B 0,C 180,E1 -19923.242,E2 -19923.242} C_VEL
LIN {X 0,Y 257.025,Z 351.539,A -85,B 0,C 180,E1 -19923.935,E2 -19923.935} C_VEL
LIN {X 0,Y 260.038,Z 311.735,A -85,B 0,C 180,E1 -19925.309,E2 -19925.309} C_VEL
LIN {X 0,Y 259.015,Z 295.622,A -85,B 0,C 180,E1 -19926.418,E2 -19926.418} C_VEL
LIN {X 0,Y 257.638,Z 282.951,A -85,B 0,C 180,E1 -19927.47,E2 -19927.47} C_VEL
LIN {X 0,Y 253.284,Z 272.362,A -85,B 0,C 180,E1 -19929.324,E2 -19929.324} C_VEL
LIN {X 0,Y 249.426,Z 264.696,A -85,B 0,C 180,E1 -19931.013,E2 -19931.013} C_VEL
LIN {X 0,Y 245.055,Z 256.622,A -85,B 0,C 180,E1 -19933.144,E2 -19933.144} C_VEL
LIN {X 0,Y 240.808,Z 249.638,A -85,B 0,C 180,E1 -19935.445,E2 -19935.445} C_VEL
LIN {X 0,Y 236.555,Z 242.859,A -85,B 0,C 180,E1 -19938.137,E2 -19938.137} C_VEL
LIN {X 0,Y 231.37,Z 235.053,A -85,B 0,C 180,E1 -19942.359,E2 -19942.359} C_VEL
LIN {X 0,Y 229.796,Z 231.323,A -85,B 0,C 180,E1 -19946.598,E2 -19946.598} C_VEL
LIN {X 0,Y 229.227,Z 229.506,A -85,B 0,C 180,E1 -19949.144,E2 -19949.144} C_VEL
LIN {X 0,Y 228.178,Z 227.364,A -85,B 0,C 180,E1 -19954.456,E2 -19954.456} C_VEL
LIN {X 0,Y 228.052,Z 226.764,A -85,B 0,C 180,E1 -19958.296,E2 -19958.296} C_VEL
LIN {X 0,Y 228.287,Z 227.371,A -85,B 0,C 180,E1 -19962.868,E2 -19962.868} C_VEL
LIN {X 0,Y 229.821,Z 229.954,A -85,B 0,C 180,E1 -19964.934,E2 -19964.934} C_VEL
LIN {X 0,Y 232.428,Z 231.755,A -85,B 0,C 180,E1 -19967.336,E2 -19967.336} C_VEL
LIN {X 0,Y 233.151,Z 232.28,A -85,B 0,C 180,E1 -19967.929,E2 -19967.929} C_VEL
LIN {X 0,Y 234.66,Z 235.154,A -85,B 0,C 180,E1 -19969.266,E2 -19969.266} C_VEL
LIN {X 0,Y 237.764,Z 237.818,A -85,B 0,C 180,E1 -19971.328,E2 -19971.328} C_VEL
LIN {X 0,Y 239.709,Z 241.025,A -85,B 0,C 180,E1 -19972.611,E2 -19972.611} C_VEL
LIN {X 0,Y 241.657,Z 243.094,A -85,B 0,C 180,E1 -19973.686,E2 -19973.686} C_VEL
LIN {X 0,Y 244.127,Z 246.63,A -85,B 0,C 180,E1 -19975.045,E2 -19975.045} C_VEL
LIN {X 0,Y 245.682,Z 248.294,A -85,B 0,C 180,E1 -19975.782,E2 -19975.782} C_VEL
LIN {X 0,Y 248.827,Z 252.769,A -85,B 0,C 180,E1 -19977.262,E2 -19977.262} C_VEL
LIN {X 0,Y 252.559,Z 258.678,A -85,B 0,C 180,E1 -19978.902,E2 -19978.902} C_VEL
LIN {X 0,Y 258.881,Z 269.633,A -85,B 0,C 180,E1 -19981.415,E2 -19981.415} C_VEL
LIN {X 0,Y 262.293,Z 276.472,A -85,B 0,C 180,E1 -19982.665,E2 -19982.665} C_VEL
LIN {X 0,Y 258.275,Z 328.571,A -85,B 0,C 180,E1 -19984.514,E2 -19984.514} C_VEL
LIN {X 0,Y 256.79,Z 341.445,A -85,B 0,C 180,E1 -19985.285,E2 -19985.285} C_VEL
LIN {X 0,Y 254.737,Z 354.06,A -85,B 0,C 180,E1 -19986.336,E2 -19986.336} C_VEL
LIN {X 0,Y 252.35,Z 365.193,A -85,B 0,C 180,E1 -19987.562,E2 -19987.562} C_VEL
LIN {X 0,Y 249.702,Z 375.386,A -85,B 0,C 180,E1 -19988.98,E2 -19988.98} C_VEL
LIN {X 0,Y 246.769,Z 385.098,A -85,B 0,C 180,E1 -19990.668,E2 -19990.668} C_VEL
LIN {X 0,Y 243.586,Z 394.196,A -85,B 0,C 180,E1 -19992.633,E2 -19992.633} C_VEL
LIN {X 0,Y 240.175,Z 402.967,A -85,B 0,C 180,E1 -19995.063,E2 -19995.063} C_VEL
LIN {X 0,Y 237.009,Z 410.29,A -85,B 0,C 180,E1 -19997.633,E2 -19997.633} C_VEL
LIN {X 0,Y 234.368,Z 415.815,A -85,B 0,C 180,E1 -20000.134,E2 -20000.134} C_VEL
LIN {X 0,Y 231.746,Z 420.85,A -85,B 0,C 180,E1 -20003.219,E2 -20003.219} C_VEL
LIN {X 0,Y 230.312,Z 423.369,A -85,B 0,C 180,E1 -20005.291,E2 -20005.291} C_VEL
LIN {X 0,Y 229.057,Z 425.229,A -85,B 0,C 180,E1 -20007.402,E2 -20007.402} C_VEL
LIN {X 0,Y 227.744,Z 426.792,A -85,B 0,C 180,E1 -20010.225,E2 -20010.225} C_VEL
LIN {X 0,Y 226.781,Z 427.308,A -85,B 0,C 180,E1 -20013.203,E2 -20013.203} C_VEL
LIN {X 0,Y 226.204,Z 426.688,A -85,B 0,C 180,E1 -20016.179,E2 -20016.179} C_VEL
LIN {X 0,Y 226.003,Z 425.067,A -85,B 0,C 180,E1 -20018.975,E2 -20018.975} C_VEL
LIN {X 0,Y 226.147,Z 422.414,A -85,B 0,C 180,E1 -20021.768,E2 -20021.768} C_VEL
LIN {X 0,Y 226.619,Z 418.749,A -85,B 0,C 180,E1 -20024.498,E2 -20024.498} C_VEL
LIN {X 0,Y 227.245,Z 414.109,A -85,B 0,C 180,E1 -20027.126,E2 -20027.126} C_VEL
LIN {X 0,Y 228.068,Z 408.425,A -85,B 0,C 180,E1 -20029.676,E2 -20029.676} C_VEL
LIN {X 0,Y 229.143,Z 401.527,A -85,B 0,C 180,E1 -20032.164,E2 -20032.164} C_VEL
LIN {X 0,Y 230.57,Z 393.069,A -85,B 0,C 180,E1 -20034.611,E2 -20034.611} C_VEL
LIN {X 0,Y 232.092,Z 382.978,A -85,B 0,C 180,E1 -20036.972,E2 -20036.972} C_VEL
LIN {X 0,Y 233.489,Z 373.717,A -85,B 0,C 180,E1 -20038.72,E2 -20038.72} C_VEL
LIN {X 0,Y 235.044,Z 361.894,A -85,B 0,C 180,E1 -20040.508,E2 -20040.508} C_VEL
LIN {X 0,Y 236.382,Z 350.33,A -85,B 0,C 180,E1 -20041.877,E2 -20041.877} C_VEL
LIN {X 0,Y 237.571,Z 337.545,A -85,B 0,C 180,E1 -20043.02,E2 -20043.02} C_VEL
LIN {X 0,Y 238.255,Z 324.298,A -85,B 0,C 180,E1 -20043.857,E2 -20043.857} C_VEL
LIN {X 0,Y 239.829,Z 288.209,A -85,B 0,C 180,E1 -20045.179,E2 -20045.179} C_VEL
LIN {X 0,Y 241.022,Z 258.729,A -85,B 0,C 180,E1 -20046.216,E2 -20046.216} C_VEL
LIN {X 0,Y 231.831,Z 235.769,A -85,B 0,C 180,E1 -20047.985,E2 -20047.985} C_VEL
LIN {X 0,Y 228.128,Z 227.052,A -85,B 0,C 180,E1 -20048.719,E2 -20048.719} C_VEL
LIN {X 0,Y 227.955,Z 226.092,A -85,B 0,C 180,E1 -20048.821,E2 -20048.821} C_VEL
LIN {X 0,Y 228.03,Z 226.08,A -85,B 0,C 180,E1 -20053.896,E2 -20053.896} C_VEL
LIN {X 0,Y 228.058,Z 226.076,A -85,B 0,C 180,E1 -20057.543,E2 -20057.543} C_VEL
LIN {X 0,Y 228.254,Z 226.053,A -85,B 0,C 180,E1 -20061.145,E2 -20061.145} C_VEL
LIN {X 0,Y 228.304,Z 226.047,A -85,B 0,C 180,E1 -20062.927,E2 -20062.927} C_VEL
LIN {X 0,Y 228.552,Z 226.015,A -85,B 0,C 180,E1 -20068.238,E2 -20068.238} C_VEL
LIN {X 0,Y 228.549,Z 226.014,A -85,B 0,C 180,E1 -20071.763,E2 -20071.763} C_VEL
LIN {X 0,Y 228.312,Z 226.043,A -85,B 0,C 180,E1 -20077.073,E2 -20077.073} C_VEL
LIN {X 0,Y 228.147,Z 226.065,A -85,B 0,C 180,E1 -20080.652,E2 -20080.652} C_VEL
LIN {X 0,Y 228.067,Z 226.077,A -85,B 0,C 180,E1 -20084.272,E2 -20084.272} C_VEL
LIN {X 0,Y 228.005,Z 226.083,A -85,B 0,C 180,E1 -20087.954,E2 -20087.954} C_VEL
LIN {X 0,Y 227.923,Z 226.084,A -85,B 0,C 180,E1 -20092.324,E2 -20092.324} C_VEL
LIN {X 0,Y 227.924,Z 226.091,A -85,B 0,C 180,E1 -20096.593,E2 -20096.593} C_VEL
LIN {X 0,Y 227.876,Z 226.098,A -85,B 0,C 180,E1 -20100.281,E2 -20100.281} C_VEL
LIN {X 0,Y 227.878,Z 226.093,A -85,B 0,C 180,E1 -20103.721,E2 -20103.721} C_VEL
LIN {X 0,Y 227.841,Z 226.085,A -85,B 0,C 180,E1 -20108.092,E2 -20108.092} C_VEL
LIN {X 0,Y 227.804,Z 226.101,A -85,B 0,C 180,E1 -20112.745,E2 -20112.745} C_VEL
LIN {X 0,Y 227.801,Z 226.11,A -85,B 0,C 180,E1 -20117.255,E2 -20117.255} C_VEL
LIN {X 0,Y 227.845,Z 226.097,A -85,B 0,C 180,E1 -20121.909,E2 -20121.909} C_VEL
LIN {X 0,Y 227.881,Z 226.096,A -85,B 0,C 180,E1 -20126.378,E2 -20126.378} C_VEL
LIN {X 0,Y 227.879,Z 226.098,A -85,B 0,C 180,E1 -20130.432,E2 -20130.432} C_VEL
LIN {X 0,Y 227.905,Z 226.089,A -85,B 0,C 180,E1 -20134.423,E2 -20134.423} C_VEL
LIN {X 0,Y 227.954,Z 226.087,A -85,B 0,C 180,E1 -20138.286,E2 -20138.286} C_VEL
LIN {X 0,Y 228.011,Z 226.081,A -85,B 0,C 180,E1 -20142.848,E2 -20142.848} C_VEL
LIN {X 0,Y 228.061,Z 226.062,A -85,B 0,C 180,E1 -20147.543,E2 -20147.543} C_VEL
LIN {X 0,Y 228.256,Z 226.034,A -85,B 0,C 180,E1 -20151.144,E2 -20151.144} C_VEL
LIN {X 0,Y 228.305,Z 226.035,A -85,B 0,C 180,E1 -20152.927,E2 -20152.927} C_VEL
LIN {X 0,Y 228.549,Z 226.015,A -85,B 0,C 180,E1 -20158.238,E2 -20158.238} C_VEL
LIN {X 0,Y 228.54,Z 226.016,A -85,B 0,C 180,E1 -20161.762,E2 -20161.762} C_VEL
LIN {X 0,Y 228.309,Z 226.032,A -85,B 0,C 180,E1 -20167.073,E2 -20167.073} C_VEL
LIN {X 0,Y 228.144,Z 226.061,A -85,B 0,C 180,E1 -20170.651,E2 -20170.651} C_VEL
LIN {X 0,Y 228.023,Z 226.083,A -85,B 0,C 180,E1 -20176.105,E2 -20176.105} C_VEL
LIN {X 0,Y 227.918,Z 226.09,A -85,B 0,C 180,E1 -20179.828,E2 -20179.828} C_VEL
LIN {X 0,Y 227.873,Z 226.099,A -85,B 0,C 180,E1 -20183.637,E2 -20183.637} C_VEL
LIN {X 0,Y 227.848,Z 226.106,A -85,B 0,C 180,E1 -20187.56,E2 -20187.56} C_VEL
LIN {X 0,Y 227.859,Z 226.099,A -85,B 0,C 180,E1 -20191.624,E2 -20191.624} C_VEL
LIN {X 0,Y 227.868,Z 226.1,A -85,B 0,C 180,E1 -20195.874,E2 -20195.874} C_VEL
LIN {X 0,Y 227.805,Z 226.109,A -85,B 0,C 180,E1 -20200.382,E2 -20200.382} C_VEL
LIN {X 0,Y 227.081,Z 226.201,A -85,B 0,C 180,E1 -20201.858,E2 -20201.858} C_VEL
LIN {X 0,Y 224.247,Z 226.552,A -85,B 0,C 180,E1 -20204.269,E2 -20204.269} C_VEL
LIN {X 0,Y 221.067,Z 226.95,A -85,B 0,C 180,E1 -20207.247,E2 -20207.247} C_VEL
LIN {X 0,Y 220.741,Z 226.987,A -85,B 0,C 180,E1 -20208.278,E2 -20208.278} C_VEL
LIN {X 0,Y 220.832,Z 227.018,A -85,B 0,C 180,E1 -20210.889,E2 -20210.889} C_VEL
LIN {X 0,Y 223.031,Z 236.915,A -85,B 0,C 180,E1 -20214.702,E2 -20214.702} C_VEL
LIN {X 0,Y 225.185,Z 247.128,A -85,B 0,C 180,E1 -20218.446,E2 -20218.446} C_VEL
LIN {X 0,Y 228.004,Z 256.651,A -85,B 0,C 180,E1 -20219.127,E2 -20219.127} C_VEL
LIN {X 0,Y 232.966,Z 308.273,A -85,B 0,C 180,E1 -20221.686,E2 -20221.686} C_VEL
LIN {X 0,Y 230.813,Z 357.92,A -85,B 0,C 180,E1 -20223.556,E2 -20223.556} C_VEL
LIN {X 0,Y 229.795,Z 371.289,A -85,B 0,C 180,E1 -20224.405,E2 -20224.405} C_VEL
LIN {X 0,Y 228.423,Z 383.04,A -85,B 0,C 180,E1 -20225.457,E2 -20225.457} C_VEL
LIN {X 0,Y 226.647,Z 395.438,A -85,B 0,C 180,E1 -20226.953,E2 -20226.953} C_VEL
LIN {X 0,Y 224.922,Z 406.659,A -85,B 0,C 180,E1 -20228.7,E2 -20228.7} C_VEL
LIN {X 0,Y 223.204,Z 416.943,A -85,B 0,C 180,E1 -20230.727,E2 -20230.727} C_VEL
LIN {X 0,Y 221.687,Z 425.996,A -85,B 0,C 180,E1 -20232.947,E2 -20232.947} C_VEL
LIN {X 0,Y 220.458,Z 434.996,A -85,B 0,C 180,E1 -20235.696,E2 -20235.696} C_VEL
LIN {X 0,Y 219.527,Z 442.104,A -85,B 0,C 180,E1 -20238.457,E2 -20238.457} C_VEL
LIN {X 0,Y 219.105,Z 448.581,A -85,B 0,C 180,E1 -20241.7,E2 -20241.7} C_VEL
LIN {X 0,Y 219.143,Z 452.762,A -85,B 0,C 180,E1 -20244.478,E2 -20244.478} C_VEL
LIN {X 0,Y 219.097,Z 454.884,A -85,B 0,C 180,E1 -20246.321,E2 -20246.321} C_VEL
LIN {X 0,Y 219.204,Z 456.515,A -85,B 0,C 180,E1 -20248.162,E2 -20248.162} C_VEL
LIN {X 0,Y 219.473,Z 457.722,A -85,B 0,C 180,E1 -20249.999,E2 -20249.999} C_VEL
LIN {X 0,Y 219.079,Z 458.433,A -85,B 0,C 180,E1 -20251.838,E2 -20251.838} C_VEL
LIN {X 0,Y 218.745,Z 458.643,A -85,B 0,C 180,E1 -20255.129,E2 -20255.129} C_VEL
LIN {X 0,Y 218.764,Z 458.035,A -85,B 0,C 180,E1 -20257.383,E2 -20257.383} C_VEL
LIN {X 0,Y 218.959,Z 457.115,A -85,B 0,C 180,E1 -20259.235,E2 -20259.235} C_VEL
LIN {X 0,Y 219.301,Z 455.777,A -85,B 0,C 180,E1 -20261.086,E2 -20261.086} C_VEL
LIN {X 0,Y 220.27,Z 453.015,A -85,B 0,C 180,E1 -20263.845,E2 -20263.845} C_VEL
LIN {X 0,Y 221.91,Z 449.267,A -85,B 0,C 180,E1 -20266.56,E2 -20266.56} C_VEL
LIN {X 0,Y 223.966,Z 444.457,A -85,B 0,C 180,E1 -20269.237,E2 -20269.237} C_VEL
LIN {X 0,Y 226.435,Z 438.465,A -85,B 0,C 180,E1 -20271.866,E2 -20271.866} C_VEL
LIN {X 0,Y 229.647,Z 431.1,A -85,B 0,C 180,E1 -20274.402,E2 -20274.402} C_VEL
LIN {X 0,Y 233.401,Z 422.076,A -85,B 0,C 180,E1 -20276.85,E2 -20276.85} C_VEL
LIN {X 0,Y 237.255,Z 411.943,A -85,B 0,C 180,E1 -20279.016,E2 -20279.016} C_VEL
LIN {X 0,Y 240.797,Z 401.724,A -85,B 0,C 180,E1 -20280.714,E2 -20280.714} C_VEL
LIN {X 0,Y 244.185,Z 390.59,A -85,B 0,C 180,E1 -20282.171,E2 -20282.171} C_VEL
LIN {X 0,Y 247.42,Z 378.381,A -85,B 0,C 180,E1 -20283.391,E2 -20283.391} C_VEL
LIN {X 0,Y 250.171,Z 364.767,A -85,B 0,C 180,E1 -20284.396,E2 -20284.396} C_VEL
LIN {X 0,Y 252.125,Z 351.124,A -85,B 0,C 180,E1 -20285.099,E2 -20285.099} C_VEL
LIN {X 0,Y 255.177,Z 312.304,A -85,B 0,C 180,E1 -20286.483,E2 -20286.483} C_VEL
LIN {X 0,Y 254.378,Z 298.27,A -85,B 0,C 180,E1 -20287.472,E2 -20287.472} C_VEL
LIN {X 0,Y 253.295,Z 286.518,A -85,B 0,C 180,E1 -20288.459,E2 -20288.459} C_VEL
LIN {X 0,Y 249.399,Z 276.868,A -85,B 0,C 180,E1 -20290.238,E2 -20290.238} C_VEL
LIN {X 0,Y 245.26,Z 268.111,A -85,B 0,C 180,E1 -20292.247,E2 -20292.247} C_VEL
LIN {X 0,Y 241.496,Z 261.357,A -85,B 0,C 180,E1 -20294.189,E2 -20294.189} C_VEL
LIN {X 0,Y 238.152,Z 255.523,A -85,B 0,C 180,E1 -20296.165,E2 -20296.165} C_VEL
LIN {X 0,Y 234.263,Z 249.036,A -85,B 0,C 180,E1 -20298.798,E2 -20298.798} C_VEL
LIN {X 0,Y 229.479,Z 241.553,A -85,B 0,C 180,E1 -20302.929,E2 -20302.929} C_VEL
LIN {X 0,Y 225.252,Z 235.561,A -85,B 0,C 180,E1 -20308.728,E2 -20308.728} C_VEL
LIN {X 0,Y 224.004,Z 233.483,A -85,B 0,C 180,E1 -20312.97,E2 -20312.97} C_VEL
LIN {X 0,Y 224.039,Z 232.928,A -85,B 0,C 180,E1 -20315.933,E2 -20315.933} C_VEL
LIN {X 0,Y 224.823,Z 233.13,A -85,B 0,C 180,E1 -20318.932,E2 -20318.932} C_VEL
LIN {X 0,Y 226.882,Z 234.417,A -85,B 0,C 180,E1 -20322.633,E2 -20322.633} C_VEL
LIN {X 0,Y 228.507,Z 237.015,A -85,B 0,C 180,E1 -20324.845,E2 -20324.845} C_VEL
LIN {X 0,Y 231.297,Z 239.027,A -85,B 0,C 180,E1 -20327.441,E2 -20327.441} C_VEL
LIN {X 0,Y 233.003,Z 242.024,A -85,B 0,C 180,E1 -20328.996,E2 -20328.996} C_VEL
LIN {X 0,Y 235.625,Z 244.382,A -85,B 0,C 180,E1 -20330.799,E2 -20330.799} C_VEL
LIN {X 0,Y 238.058,Z 248.06,A -85,B 0,C 180,E1 -20332.441,E2 -20332.441} C_VEL
LIN {X 0,Y 239.347,Z 249.593,A -85,B 0,C 180,E1 -20333.182,E2 -20333.182} C_VEL
LIN {X 0,Y 242.118,Z 253.332,A -85,B 0,C 180,E1 -20334.73,E2 -20334.73} C_VEL
LIN {X 0,Y 243.535,Z 255.246,A -85,B 0,C 180,E1 -20335.47,E2 -20335.47} C_VEL
LIN {X 0,Y 246.355,Z 259.323,A -85,B 0,C 180,E1 -20336.833,E2 -20336.833} C_VEL
LIN {X 0,Y 249.917,Z 265.473,A -85,B 0,C 180,E1 -20338.504,E2 -20338.504} C_VEL
LIN {X 0,Y 255.204,Z 274.767,A -85,B 0,C 180,E1 -20340.687,E2 -20340.687} C_VEL
LIN {X 0,Y 257.397,Z 279.293,A -85,B 0,C 180,E1 -20341.564,E2 -20341.564} C_VEL
LIN {X 0,Y 253.387,Z 329.398,A -85,B 0,C 180,E1 -20343.378,E2 -20343.378} C_VEL
LIN {X 0,Y 251.943,Z 341.379,A -85,B 0,C 180,E1 -20344.098,E2 -20344.098} C_VEL
LIN {X 0,Y 249.721,Z 354.451,A -85,B 0,C 180,E1 -20345.197,E2 -20345.197} C_VEL
LIN {X 0,Y 246.98,Z 366.368,A -85,B 0,C 180,E1 -20346.536,E2 -20346.536} C_VEL
LIN {X 0,Y 244.017,Z 377.018,A -85,B 0,C 180,E1 -20348.071,E2 -20348.071} C_VEL
LIN {X 0,Y 240.906,Z 386.643,A -85,B 0,C 180,E1 -20349.798,E2 -20349.798} C_VEL
LIN {X 0,Y 237.334,Z 396.167,A -85,B 0,C 180,E1 -20351.963,E2 -20351.963} C_VEL
LIN {X 0,Y 233.722,Z 404.777,A -85,B 0,C 180,E1 -20354.464,E2 -20354.464} C_VEL
LIN {X 0,Y 230.734,Z 411.148,A -85,B 0,C 180,E1 -20356.82,E2 -20356.82} C_VEL
LIN {X 0,Y 228.416,Z 415.637,A -85,B 0,C 180,E1 -20358.897,E2 -20358.897} C_VEL
LIN {X 0,Y 225.618,Z 420.783,A -85,B 0,C 180,E1 -20361.95,E2 -20361.95} C_VEL
LIN {X 0,Y 223.78,Z 423.759,A -85,B 0,C 180,E1 -20364.389,E2 -20364.389} C_VEL
LIN {X 0,Y 221.893,Z 426.358,A -85,B 0,C 180,E1 -20367.522,E2 -20367.522} C_VEL
LIN {X 0,Y 220.474,Z 427.669,A -85,B 0,C 180,E1 -20370.666,E2 -20370.666} C_VEL
LIN {X 0,Y 219.575,Z 427.805,A -85,B 0,C 180,E1 -20373.676,E2 -20373.676} C_VEL
LIN {X 0,Y 219.053,Z 426.867,A -85,B 0,C 180,E1 -20376.671,E2 -20376.671} C_VEL
LIN {X 0,Y 218.917,Z 424.595,A -85,B 0,C 180,E1 -20379.946,E2 -20379.946} C_VEL
LIN {X 0,Y 219.378,Z 420.531,A -85,B 0,C 180,E1 -20383.54,E2 -20383.54} C_VEL
LIN {X 0,Y 219.897,Z 416.374,A -85,B 0,C 180,E1 -20386.181,E2 -20386.181} C_VEL
LIN {X 0,Y 220.815,Z 410.046,A -85,B 0,C 180,E1 -20389.269,E2 -20389.269} C_VEL
LIN {X 0,Y 221.919,Z 403.046,A -85,B 0,C 180,E1 -20391.964,E2 -20391.964} C_VEL
LIN {X 0,Y 223.318,Z 394.852,A -85,B 0,C 180,E1 -20394.498,E2 -20394.498} C_VEL
LIN {X 0,Y 224.94,Z 384.473,A -85,B 0,C 180,E1 -20397.055,E2 -20397.055} C_VEL
LIN {X 0,Y 226.567,Z 374.191,A -85,B 0,C 180,E1 -20399.08,E2 -20399.08} C_VEL
LIN {X 0,Y 228.078,Z 363.042,A -85,B 0,C 180,E1 -20400.829,E2 -20400.829} C_VEL
LIN {X 0,Y 229.579,Z 350.497,A -85,B 0,C 180,E1 -20402.364,E2 -20402.364} C_VEL
LIN {X 0,Y 230.643,Z 339.243,A -85,B 0,C 180,E1 -20403.414,E2 -20403.414} C_VEL
LIN {X 0,Y 231.473,Z 325.417,A -85,B 0,C 180,E1 -20404.334,E2 -20404.334} C_VEL
LIN {X 0,Y 232.638,Z 299.259,A -85,B 0,C 180,E1 -20405.357,E2 -20405.357} C_VEL
LIN {X 0,Y 234.248,Z 260.141,A -85,B 0,C 180,E1 -20406.776,E2 -20406.776} C_VEL
LIN {X 0,Y 225.173,Z 237.602,A -85,B 0,C 180,E1 -20408.576,E2 -20408.576} C_VEL
LIN {X 0,Y 220.961,Z 227.304,A -85,B 0,C 180,E1 -20409.46,E2 -20409.46} C_VEL
LIN {X 0,Y 220.904,Z 226.969,A -85,B 0,C 180,E1 -20409.515,E2 -20409.515} C_VEL
LIN {X 0,Y 221,Z 226.957,A -85,B 0,C 180,E1 -20413.369,E2 -20413.369} C_VEL
LIN {X 0,Y 221.063,Z 226.95,A -85,B 0,C 180,E1 -20419.004,E2 -20419.004} C_VEL
LIN {X 0,Y 221.241,Z 226.928,A -85,B 0,C 180,E1 -20422.7,E2 -20422.7} C_VEL
LIN {X 0,Y 221.51,Z 226.892,A -85,B 0,C 180,E1 -20428.182,E2 -20428.182} C_VEL
LIN {X 0,Y 221.506,Z 226.891,A -85,B 0,C 180,E1 -20431.819,E2 -20431.819} C_VEL
LIN {X 0,Y 221.248,Z 226.923,A -85,B 0,C 180,E1 -20437.3,E2 -20437.3} C_VEL
LIN {X 0,Y 221.069,Z 226.946,A -85,B 0,C 180,E1 -20440.997,E2 -20440.997} C_VEL
LIN {X 0,Y 220.998,Z 226.955,A -85,B 0,C 180,E1 -20444.739,E2 -20444.739} C_VEL
LIN {X 0,Y 220.922,Z 226.961,A -85,B 0,C 180,E1 -20448.55,E2 -20448.55} C_VEL
LIN {X 0,Y 220.87,Z 226.962,A -85,B 0,C 180,E1 -20452.666,E2 -20452.666} C_VEL
LIN {X 0,Y 220.867,Z 226.97,A -85,B 0,C 180,E1 -20457.006,E2 -20457.006} C_VEL
LIN {X 0,Y 220.82,Z 226.976,A -85,B 0,C 180,E1 -20460.759,E2 -20460.759} C_VEL
LIN {X 0,Y 220.795,Z 226.971,A -85,B 0,C 180,E1 -20464.957,E2 -20464.957} C_VEL
LIN {X 0,Y 220.803,Z 226.962,A -85,B 0,C 180,E1 -20467.276,E2 -20467.276} C_VEL
LIN {X 0,Y 220.763,Z 226.979,A -85,B 0,C 180,E1 -20471.955,E2 -20471.955} C_VEL
LIN {X 0,Y 220.767,Z 226.986,A -85,B 0,C 180,E1 -20475.544,E2 -20475.544} C_VEL
LIN {X 0,Y 220.785,Z 226.979,A -85,B 0,C 180,E1 -20480.459,E2 -20480.459} C_VEL
LIN {X 0,Y 220.827,Z 226.972,A -85,B 0,C 180,E1 -20482.793,E2 -20482.793} C_VEL
LIN {X 0,Y 220.814,Z 226.981,A -85,B 0,C 180,E1 -20487.244,E2 -20487.244} C_VEL
LIN {X 0,Y 220.806,Z 226.977,A -85,B 0,C 180,E1 -20491.482,E2 -20491.482} C_VEL
LIN {X 0,Y 220.85,Z 226.969,A -85,B 0,C 180,E1 -20495.563,E2 -20495.563} C_VEL
LIN {X 0,Y 220.881,Z 226.969,A -85,B 0,C 180,E1 -20499.513,E2 -20499.513} C_VEL
LIN {X 0,Y 220.994,Z 226.952,A -85,B 0,C 180,E1 -20503.369,E2 -20503.369} C_VEL
LIN {X 0,Y 221.065,Z 226.926,A -85,B 0,C 180,E1 -20509.004,E2 -20509.004} C_VEL
LIN {X 0,Y 221.242,Z 226.911,A -85,B 0,C 180,E1 -20512.7,E2 -20512.7} C_VEL
LIN {X 0,Y 221.507,Z 226.892,A -85,B 0,C 180,E1 -20518.182,E2 -20518.182} C_VEL
LIN {X 0,Y 221.473,Z 226.896,A -85,B 0,C 180,E1 -20521.819,E2 -20521.819} C_VEL
LIN {X 0,Y 221.246,Z 226.911,A -85,B 0,C 180,E1 -20527.3,E2 -20527.3} C_VEL
LIN {X 0,Y 221.064,Z 226.942,A -85,B 0,C 180,E1 -20530.997,E2 -20530.997} C_VEL
LIN {X 0,Y 220.981,Z 226.958,A -85,B 0,C 180,E1 -20536.633,E2 -20536.633} C_VEL
LIN {X 0,Y 220.872,Z 226.963,A -85,B 0,C 180,E1 -20540.488,E2 -20540.488} C_VEL
LIN {X 0,Y 220.808,Z 226.98,A -85,B 0,C 180,E1 -20544.442,E2 -20544.442} C_VEL
LIN {X 0,Y 220.802,Z 226.979,A -85,B 0,C 180,E1 -20548.519,E2 -20548.519} C_VEL
LIN {X 0,Y 220.815,Z 226.977,A -85,B 0,C 180,E1 -20552.757,E2 -20552.757} C_VEL
LIN {X 0,Y 220.804,Z 226.981,A -85,B 0,C 180,E1 -20557.275,E2 -20557.275} C_VEL
LIN {X 0,Y 220.752,Z 226.988,A -85,B 0,C 180,E1 -20561.957,E2 -20561.957} C_VEL
LIN {X 0,Y 220.755,Z 226.988,A -85,B 0,C 180,E1 -20565.54,E2 -20565.54} C_VEL
LIN {X 0,Y 220.741,Z 226.987,A -85,B 0,C 180,E1 -20568.278,E2 -20568.278} C_VEL
LIN {X 0,Y 220.477,Z 227.377,A -85,B 0,C 180,E1 -20569.283,E2 -20569.283} C_VEL
LIN {X 0,Y 219.484,Z 229.121,A -85,B 0,C 180,E1 -20570.725,E2 -20570.725} C_VEL
LIN {X 0,Y 218.208,Z 231.803,A -85,B 0,C 180,E1 -20572.075,E2 -20572.075} C_VEL
LIN {X 0,Y 216.755,Z 236.316,A -85,B 0,C 180,E1 -20573.832,E2 -20573.832} C_VEL
LIN {X 0,Y 216.487,Z 239.898,A -85,B 0,C 180,E1 -20575.139,E2 -20575.139} C_VEL
LIN {X 0,Y 216.654,Z 241.063,A -85,B 0,C 180,E1 -20575.578,E2 -20575.578} C_VEL
LIN {X 0,Y 217.817,Z 246.596,A -85,B 0,C 180,E1 -20577.665,E2 -20577.665} C_VEL
LIN {X 0,Y 221.436,Z 257.959,A -85,B 0,C 180,E1 -20578.534,E2 -20578.534} C_VEL
LIN {X 0,Y 226.246,Z 308.437,A -85,B 0,C 180,E1 -20581.116,E2 -20581.116} C_VEL
LIN {X 0,Y 224.045,Z 357.106,A -85,B 0,C 180,E1 -20583.007,E2 -20583.007} C_VEL
LIN {X 0,Y 223.031,Z 370.551,A -85,B 0,C 180,E1 -20583.884,E2 -20583.884} C_VEL
LIN {X 0,Y 221.542,Z 382.831,A -85,B 0,C 180,E1 -20585.019,E2 -20585.019} C_VEL
LIN {X 0,Y 219.626,Z 395.932,A -85,B 0,C 180,E1 -20586.671,E2 -20586.671} C_VEL
LIN {X 0,Y 217.868,Z 406.938,A -85,B 0,C 180,E1 -20588.473,E2 -20588.473} C_VEL
LIN {X 0,Y 216.111,Z 417.099,A -85,B 0,C 180,E1 -20590.578,E2 -20590.578} C_VEL
LIN {X 0,Y 214.585,Z 425.98,A -85,B 0,C 180,E1 -20592.856,E2 -20592.856} C_VEL
LIN {X 0,Y 213.367,Z 434.871,A -85,B 0,C 180,E1 -20595.697,E2 -20595.697} C_VEL
LIN {X 0,Y 212.437,Z 441.885,A -85,B 0,C 180,E1 -20598.55,E2 -20598.55} C_VEL
LIN {X 0,Y 212.06,Z 447.475,A -85,B 0,C 180,E1 -20601.423,E2 -20601.423} C_VEL
LIN {X 0,Y 212.069,Z 451.79,A -85,B 0,C 180,E1 -20604.294,E2 -20604.294} C_VEL
LIN {X 0,Y 212.038,Z 454.013,A -85,B 0,C 180,E1 -20606.199,E2 -20606.199} C_VEL
LIN {X 0,Y 212.125,Z 455.727,A -85,B 0,C 180,E1 -20608.101,E2 -20608.101} C_VEL
LIN {X 0,Y 212.414,Z 456.993,A -85,B 0,C 180,E1 -20609.999,E2 -20609.999} C_VEL
LIN {X 0,Y 211.838,Z 458.132,A -85,B 0,C 180,E1 -20613.804,E2 -20613.804} C_VEL
LIN {X 0,Y 211.685,Z 457.575,A -85,B 0,C 180,E1 -20617.631,E2 -20617.631} C_VEL
LIN {X 0,Y 212.294,Z 455.471,A -85,B 0,C 180,E1 -20621.456,E2 -20621.456} C_VEL
LIN {X 0,Y 213.353,Z 452.808,A -85,B 0,C 180,E1 -20624.303,E2 -20624.303} C_VEL
LIN {X 0,Y 215.065,Z 449.181,A -85,B 0,C 180,E1 -20627.103,E2 -20627.103} C_VEL
LIN {X 0,Y 217.587,Z 443.7,A -85,B 0,C 180,E1 -20630.298,E2 -20630.298} C_VEL
LIN {X 0,Y 220.36,Z 437.665,A -85,B 0,C 180,E1 -20632.997,E2 -20632.997} C_VEL
LIN {X 0,Y 223.862,Z 430.256,A -85,B 0,C 180,E1 -20635.573,E2 -20635.573} C_VEL
LIN {X 0,Y 227.894,Z 421.164,A -85,B 0,C 180,E1 -20638.053,E2 -20638.053} C_VEL
LIN {X 0,Y 231.921,Z 410.971,A -85,B 0,C 180,E1 -20640.251,E2 -20640.251} C_VEL
LIN {X 0,Y 236.089,Z 399.485,A -85,B 0,C 180,E1 -20642.148,E2 -20642.148} C_VEL
LIN {X 0,Y 239.693,Z 388.092,A -85,B 0,C 180,E1 -20643.602,E2 -20643.602} C_VEL
LIN {X 0,Y 243.107,Z 375.243,A -85,B 0,C 180,E1 -20644.816,E2 -20644.816} C_VEL
LIN {X 0,Y 245.77,Z 361.884,A -85,B 0,C 180,E1 -20645.762,E2 -20645.762} C_VEL
LIN {X 0,Y 247.599,Z 348.545,A -85,B 0,C 180,E1 -20646.399,E2 -20646.399} C_VEL
LIN {X 0,Y 250.473,Z 313.583,A -85,B 0,C 180,E1 -20647.653,E2 -20647.653} C_VEL
LIN {X 0,Y 249.857,Z 300.098,A -85,B 0,C 180,E1 -20648.646,E2 -20648.646} C_VEL
LIN {X 0,Y 248.995,Z 289.94,A -85,B 0,C 180,E1 -20649.533,E2 -20649.533} C_VEL
LIN {X 0,Y 245.632,Z 281.409,A -85,B 0,C 180,E1 -20651.176,E2 -20651.176} C_VEL
LIN {X 0,Y 241.941,Z 273.266,A -85,B 0,C 180,E1 -20653.112,E2 -20653.112} C_VEL
LIN {X 0,Y 238.681,Z 267.088,A -85,B 0,C 180,E1 -20654.944,E2 -20654.944} C_VEL
LIN {X 0,Y 235.584,Z 261.494,A -85,B 0,C 180,E1 -20656.869,E2 -20656.869} C_VEL
LIN {X 0,Y 231.996,Z 255.207,A -85,B 0,C 180,E1 -20659.484,E2 -20659.484} C_VEL
LIN {X 0,Y 227.67,Z 248.124,A -85,B 0,C 180,E1 -20663.477,E2 -20663.477} C_VEL
LIN {X 0,Y 223.919,Z 242.445,A -85,B 0,C 180,E1 -20669.028,E2 -20669.028} C_VEL
LIN {X 0,Y 222.78,Z 240.334,A -85,B 0,C 180,E1 -20673.474,E2 -20673.474} C_VEL
LIN {X 0,Y 222.888,Z 239.91,A -85,B 0,C 180,E1 -20676.122,E2 -20676.122} C_VEL
LIN {X 0,Y 224.022,Z 240.335,A -85,B 0,C 180,E1 -20679.812,E2 -20679.812} C_VEL
LIN {X 0,Y 225.454,Z 241.354,A -85,B 0,C 180,E1 -20682.34,E2 -20682.34} C_VEL
LIN {X 0,Y 227.363,Z 244.179,A -85,B 0,C 180,E1 -20684.939,E2 -20684.939} C_VEL
LIN {X 0,Y 229.515,Z 245.776,A -85,B 0,C 180,E1 -20686.987,E2 -20686.987} C_VEL
LIN {X 0,Y 231.398,Z 248.923,A -85,B 0,C 180,E1 -20688.753,E2 -20688.753} C_VEL
LIN {X 0,Y 233.612,Z 251.072,A -85,B 0,C 180,E1 -20690.336,E2 -20690.336} C_VEL
LIN {X 0,Y 236.236,Z 254.89,A -85,B 0,C 180,E1 -20692.166,E2 -20692.166} C_VEL
LIN {X 0,Y 239.893,Z 259.827,A -85,B 0,C 180,E1 -20694.299,E2 -20694.299} C_VEL
LIN {X 0,Y 243.228,Z 264.841,A -85,B 0,C 180,E1 -20696.07,E2 -20696.07} C_VEL
LIN {X 0,Y 246.373,Z 270.293,A -85,B 0,C 180,E1 -20697.616,E2 -20697.616} C_VEL
LIN {X 0,Y 251.646,Z 279.984,A -85,B 0,C 180,E1 -20699.957,E2 -20699.957} C_VEL
LIN {X 0,Y 252.799,Z 282.393,A -85,B 0,C 180,E1 -20700.448,E2 -20700.448} C_VEL
LIN {X 0,Y 248.723,Z 329.201,A -85,B 0,C 180,E1 -20702.145,E2 -20702.145} C_VEL
LIN {X 0,Y 247.016,Z 342.69,A -85,B 0,C 180,E1 -20702.968,E2 -20702.968} C_VEL
LIN {X 0,Y 244.76,Z 355.172,A -85,B 0,C 180,E1 -20704.034,E2 -20704.034} C_VEL
LIN {X 0,Y 241.795,Z 367.437,A -85,B 0,C 180,E1 -20705.434,E2 -20705.434} C_VEL
LIN {X 0,Y 238.692,Z 377.963,A -85,B 0,C 180,E1 -20706.976,E2 -20706.976} C_VEL
LIN {X 0,Y 235.318,Z 387.735,A -85,B 0,C 180,E1 -20708.785,E2 -20708.785} C_VEL
LIN {X 0,Y 231.739,Z 396.596,A -85,B 0,C 180,E1 -20710.84,E2 -20710.84} C_VEL
LIN {X 0,Y 227.954,Z 405.173,A -85,B 0,C 180,E1 -20713.369,E2 -20713.369} C_VEL
LIN {X 0,Y 224.936,Z 411.247,A -85,B 0,C 180,E1 -20715.631,E2 -20715.631} C_VEL
LIN {X 0,Y 221.648,Z 417.245,A -85,B 0,C 180,E1 -20718.486,E2 -20718.486} C_VEL
LIN {X 0,Y 218.909,Z 421.77,A -85,B 0,C 180,E1 -20721.404,E2 -20721.404} C_VEL
LIN {X 0,Y 216.261,Z 425.602,A -85,B 0,C 180,E1 -20724.991,E2 -20724.991} C_VEL
LIN {X 0,Y 214.61,Z 427.465,A -85,B 0,C 180,E1 -20727.849,E2 -20727.849} C_VEL
LIN {X 0,Y 213.262,Z 428.406,A -85,B 0,C 180,E1 -20731.039,E2 -20731.039} C_VEL
LIN {X 0,Y 212.377,Z 428.191,A -85,B 0,C 180,E1 -20734.233,E2 -20734.233} C_VEL
LIN {X 0,Y 211.924,Z 426.928,A -85,B 0,C 180,E1 -20737.259,E2 -20737.259} C_VEL
LIN {X 0,Y 211.856,Z 424.638,A -85,B 0,C 180,E1 -20740.272,E2 -20740.272} C_VEL
LIN {X 0,Y 212.207,Z 421.317,A -85,B 0,C 180,E1 -20743.231,E2 -20743.231} C_VEL
LIN {X 0,Y 212.899,Z 416.119,A -85,B 0,C 180,E1 -20746.572,E2 -20746.572} C_VEL
LIN {X 0,Y 213.858,Z 409.607,A -85,B 0,C 180,E1 -20749.753,E2 -20749.753} C_VEL
LIN {X 0,Y 214.98,Z 402.834,A -85,B 0,C 180,E1 -20752.369,E2 -20752.369} C_VEL
LIN {X 0,Y 216.392,Z 394.64,A -85,B 0,C 180,E1 -20754.921,E2 -20754.921} C_VEL
LIN {X 0,Y 218.051,Z 384.404,A -85,B 0,C 180,E1 -20757.487,E2 -20757.487} C_VEL
LIN {X 0,Y 219.669,Z 374.397,A -85,B 0,C 180,E1 -20759.495,E2 -20759.495} C_VEL
LIN {X 0,Y 221.378,Z 362.172,A -85,B 0,C 180,E1 -20761.434,E2 -20761.434} C_VEL
LIN {X 0,Y 222.822,Z 350.188,A -85,B 0,C 180,E1 -20762.912,E2 -20762.912} C_VEL
LIN {X 0,Y 224.081,Z 336.892,A -85,B 0,C 180,E1 -20764.12,E2 -20764.12} C_VEL
LIN {X 0,Y 224.76,Z 324.799,A -85,B 0,C 180,E1 -20764.907,E2 -20764.907} C_VEL
LIN {X 0,Y 227.646,Z 261.975,A -85,B 0,C 180,E1 -20767.307,E2 -20767.307} C_VEL
LIN {X 0,Y 218.432,Z 239.173,A -85,B 0,C 180,E1 -20769.211,E2 -20769.211} C_VEL
LIN {X 0,Y 213.911,Z 228.234,A -85,B 0,C 180,E1 -20770.196,E2 -20770.196} C_VEL
LIN {X 0,Y 213.836,Z 227.849,A -85,B 0,C 180,E1 -20770.314,E2 -20770.314} C_VEL
LIN {X 0,Y 213.92,Z 227.839,A -85,B 0,C 180,E1 -20772.802,E2 -20772.802} C_VEL
LIN {X 0,Y 213.938,Z 227.838,A -85,B 0,C 180,E1 -20776.706,E2 -20776.706} C_VEL
LIN {X 0,Y 214.135,Z 227.813,A -85,B 0,C 180,E1 -20780.555,E2 -20780.555} C_VEL
LIN {X 0,Y 214.087,Z 227.818,A -85,B 0,C 180,E1 -20784.349,E2 -20784.349} C_VEL
LIN {X 0,Y 214.443,Z 227.772,A -85,B 0,C 180,E1 -20788.122,E2 -20788.122} C_VEL
LIN {X 0,Y 214.543,Z 227.759,A -85,B 0,C 180,E1 -20790.001,E2 -20790.001} C_VEL
LIN {X 0,Y 214.439,Z 227.772,A -85,B 0,C 180,E1 -20791.879,E2 -20791.879} C_VEL
LIN {X 0,Y 214.189,Z 227.802,A -85,B 0,C 180,E1 -20797.542,E2 -20797.542} C_VEL
LIN {X 0,Y 214.001,Z 227.826,A -85,B 0,C 180,E1 -20801.365,E2 -20801.365} C_VEL
LIN {X 0,Y 213.936,Z 227.835,A -85,B 0,C 180,E1 -20805.237,E2 -20805.237} C_VEL
LIN {X 0,Y 213.839,Z 227.843,A -85,B 0,C 180,E1 -20809.188,E2 -20809.188} C_VEL
LIN {X 0,Y 213.805,Z 227.841,A -85,B 0,C 180,E1 -20813.233,E2 -20813.233} C_VEL
LIN {X 0,Y 213.789,Z 227.853,A -85,B 0,C 180,E1 -20817.429,E2 -20817.429} C_VEL
LIN {X 0,Y 213.76,Z 227.856,A -85,B 0,C 180,E1 -20821.739,E2 -20821.739} C_VEL
LIN {X 0,Y 213.743,Z 227.841,A -85,B 0,C 180,E1 -20826.289,E2 -20826.289} C_VEL
LIN {X 0,Y 213.706,Z 227.852,A -85,B 0,C 180,E1 -20831.128,E2 -20831.128} C_VEL
LIN {X 0,Y 213.704,Z 227.862,A -85,B 0,C 180,E1 -20833.68,E2 -20833.68} C_VEL
LIN {X 0,Y 213.704,Z 227.863,A -85,B 0,C 180,E1 -20836.345,E2 -20836.345} C_VEL
LIN {X 0,Y 213.711,Z 227.861,A -85,B 0,C 180,E1 -20841.331,E2 -20841.331} C_VEL
LIN {X 0,Y 213.758,Z 227.855,A -85,B 0,C 180,E1 -20846.018,E2 -20846.018} C_VEL
LIN {X 0,Y 213.752,Z 227.857,A -85,B 0,C 180,E1 -20850.45,E2 -20850.45} C_VEL
LIN {X 0,Y 213.784,Z 227.848,A -85,B 0,C 180,E1 -20854.7,E2 -20854.7} C_VEL
LIN {X 0,Y 213.803,Z 227.853,A -85,B 0,C 180,E1 -20858.803,E2 -20858.803} C_VEL
LIN {X 0,Y 213.924,Z 227.835,A -85,B 0,C 180,E1 -20862.802,E2 -20862.802} C_VEL
LIN {X 0,Y 213.94,Z 227.822,A -85,B 0,C 180,E1 -20866.706,E2 -20866.706} C_VEL
LIN {X 0,Y 214.136,Z 227.787,A -85,B 0,C 180,E1 -20870.555,E2 -20870.555} C_VEL
LIN {X 0,Y 214.083,Z 227.807,A -85,B 0,C 180,E1 -20874.348,E2 -20874.348} C_VEL
LIN {X 0,Y 214.44,Z 227.772,A -85,B 0,C 180,E1 -20878.122,E2 -20878.122} C_VEL
LIN {X 0,Y 214.518,Z 227.763,A -85,B 0,C 180,E1 -20880,E2 -20880} C_VEL
LIN {X 0,Y 214.41,Z 227.776,A -85,B 0,C 180,E1 -20881.879,E2 -20881.879} C_VEL
LIN {X 0,Y 214.188,Z 227.79,A -85,B 0,C 180,E1 -20887.542,E2 -20887.542} C_VEL
LIN {X 0,Y 213.995,Z 227.823,A -85,B 0,C 180,E1 -20891.365,E2 -20891.365} C_VEL
LIN {X 0,Y 213.9,Z 227.841,A -85,B 0,C 180,E1 -20895.24,E2 -20895.24} C_VEL
LIN {X 0,Y 213.814,Z 227.847,A -85,B 0,C 180,E1 -20899.19,E2 -20899.19} C_VEL
LIN {X 0,Y 213.789,Z 227.851,A -85,B 0,C 180,E1 -20903.234,E2 -20903.234} C_VEL
LIN {X 0,Y 213.787,Z 227.857,A -85,B 0,C 180,E1 -20907.426,E2 -20907.426} C_VEL
LIN {X 0,Y 213.761,Z 227.855,A -85,B 0,C 180,E1 -20911.739,E2 -20911.739} C_VEL
LIN {X 0,Y 213.744,Z 227.858,A -85,B 0,C 180,E1 -20916.289,E2 -20916.289} C_VEL
LIN {X 0,Y 213.701,Z 227.869,A -85,B 0,C 180,E1 -20921.128,E2 -20921.128} C_VEL
LIN {X 0,Y 213.703,Z 227.867,A -85,B 0,C 180,E1 -20923.68,E2 -20923.68} C_VEL
LIN {X 0,Y 213.664,Z 227.866,A -85,B 0,C 180,E1 -20928.299,E2 -20928.299} C_VEL
LIN {X 0,Y 213.752,Z 227.919,A -85,B 0,C 180,E1 -20930.38,E2 -20930.38} C_VEL
LIN {X 0,Y 216.031,Z 238.054,A -85,B 0,C 180,E1 -20934.421,E2 -20934.421} C_VEL
LIN {X 0,Y 216.654,Z 241.063,A -85,B 0,C 180,E1 -20935.578,E2 -20935.578} C_VEL
LIN {X 0,Y 216.95,Z 243.679,A -85,B 0,C 180,E1 -20936.332,E2 -20936.332} C_VEL
LIN {X 0,Y 216.969,Z 246.882,A -85,B 0,C 180,E1 -20936.921,E2 -20936.921} C_VEL
LIN {X 0,Y 216.659,Z 252.331,A -85,B 0,C 180,E1 -20937.551,E2 -20937.551} C_VEL
LIN {X 0,Y 215.884,Z 262.417,A -85,B 0,C 180,E1 -20938.158,E2 -20938.158} C_VEL
LIN {X 0,Y 215.904,Z 270.674,A -85,B 0,C 180,E1 -20938.535,E2 -20938.535} C_VEL
LIN {X 0,Y 219.5,Z 309.612,A -85,B 0,C 180,E1 -20940.579,E2 -20940.579} C_VEL
LIN {X 0,Y 217.242,Z 356.918,A -85,B 0,C 180,E1 -20942.482,E2 -20942.482} C_VEL
LIN {X 0,Y 216.26,Z 369.531,A -85,B 0,C 180,E1 -20943.328,E2 -20943.328} C_VEL
LIN {X 0,Y 214.679,Z 382.46,A -85,B 0,C 180,E1 -20944.552,E2 -20944.552} C_VEL
LIN {X 0,Y 212.851,Z 394.753,A -85,B 0,C 180,E1 -20946.141,E2 -20946.141} C_VEL
LIN {X 0,Y 211.029,Z 405.894,A -85,B 0,C 180,E1 -20947.996,E2 -20947.996} C_VEL
LIN {X 0,Y 209.199,Z 416.15,A -85,B 0,C 180,E1 -20950.162,E2 -20950.162} C_VEL
LIN {X 0,Y 207.484,Z 425.941,A -85,B 0,C 180,E1 -20952.759,E2 -20952.759} C_VEL
LIN {X 0,Y 206.422,Z 433.386,A -85,B 0,C 180,E1 -20955.205,E2 -20955.205} C_VEL
LIN {X 0,Y 205.429,Z 440.629,A -85,B 0,C 180,E1 -20958.154,E2 -20958.154} C_VEL
LIN {X 0,Y 205.012,Z 446.367,A -85,B 0,C 180,E1 -20961.125,E2 -20961.125} C_VEL
LIN {X 0,Y 205.009,Z 450.82,A -85,B 0,C 180,E1 -20964.096,E2 -20964.096} C_VEL
LIN {X 0,Y 204.982,Z 453.108,A -85,B 0,C 180,E1 -20966.067,E2 -20966.067} C_VEL
LIN {X 0,Y 205.048,Z 454.93,A -85,B 0,C 180,E1 -20968.035,E2 -20968.035} C_VEL
LIN {X 0,Y 205.356,Z 456.263,A -85,B 0,C 180,E1 -20969.999,E2 -20969.999} C_VEL
LIN {X 0,Y 204.761,Z 457.506,A -85,B 0,C 180,E1 -20973.936,E2 -20973.936} C_VEL
LIN {X 0,Y 204.567,Z 457.525,A -85,B 0,C 180,E1 -20975.915,E2 -20975.915} C_VEL
LIN {X 0,Y 204.622,Z 457.123,A -85,B 0,C 180,E1 -20977.896,E2 -20977.896} C_VEL
LIN {X 0,Y 205.305,Z 455.138,A -85,B 0,C 180,E1 -20981.852,E2 -20981.852} C_VEL
LIN {X 0,Y 205.945,Z 453.562,A -85,B 0,C 180,E1 -20983.82,E2 -20983.82} C_VEL
LIN {X 0,Y 207.632,Z 450.409,A -85,B 0,C 180,E1 -20986.72,E2 -20986.72} C_VEL
LIN {X 0,Y 210.263,Z 445.267,A -85,B 0,C 180,E1 -20990.169,E2 -20990.169} C_VEL
LIN {X 0,Y 212.791,Z 440.059,A -85,B 0,C 180,E1 -20992.834,E2 -20992.834} C_VEL
LIN {X 0,Y 216.212,Z 433.334,A -85,B 0,C 180,E1 -20995.511,E2 -20995.511} C_VEL
LIN {X 0,Y 220.226,Z 425.128,A -85,B 0,C 180,E1 -20998.08,E2 -20998.08} C_VEL
LIN {X 0,Y 224.688,Z 415.093,A -85,B 0,C 180,E1 -21000.549,E2 -21000.549} C_VEL
LIN {X 0,Y 228.86,Z 404.711,A -85,B 0,C 180,E1 -21002.506,E2 -21002.506} C_VEL
LIN {X 0,Y 232.912,Z 393.222,A -85,B 0,C 180,E1 -21004.194,E2 -21004.194} C_VEL
LIN {X 0,Y 236.347,Z 382.067,A -85,B 0,C 180,E1 -21005.44,E2 -21005.44} C_VEL
LIN {X 0,Y 239.688,Z 368.647,A -85,B 0,C 180,E1 -21006.554,E2 -21006.554} C_VEL
LIN {X 0,Y 242.144,Z 355.33,A -85,B 0,C 180,E1 -21007.357,E2 -21007.357} C_VEL
LIN {X 0,Y 243.852,Z 339.601,A -85,B 0,C 180,E1 -21007.996,E2 -21007.996} C_VEL
LIN {X 0,Y 246.008,Z 314.74,A -85,B 0,C 180,E1 -21008.893,E2 -21008.893} C_VEL
LIN {X 0,Y 245.505,Z 302.254,A -85,B 0,C 180,E1 -21009.84,E2 -21009.84} C_VEL
LIN {X 0,Y 244.802,Z 293.394,A -85,B 0,C 180,E1 -21010.642,E2 -21010.642} C_VEL
LIN {X 0,Y 241.62,Z 285.016,A -85,B 0,C 180,E1 -21012.364,E2 -21012.364} C_VEL
LIN {X 0,Y 238.409,Z 277.885,A -85,B 0,C 180,E1 -21014.166,E2 -21014.166} C_VEL
LIN {X 0,Y 235.608,Z 272.24,A -85,B 0,C 180,E1 -21015.9,E2 -21015.9} C_VEL
LIN {X 0,Y 232.97,Z 267.24,A -85,B 0,C 180,E1 -21017.682,E2 -21017.682} C_VEL
LIN {X 0,Y 229.81,Z 261.421,A -85,B 0,C 180,E1 -21020.149,E2 -21020.149} C_VEL
LIN {X 0,Y 225.95,Z 254.736,A -85,B 0,C 180,E1 -21023.97,E2 -21023.97} C_VEL
LIN {X 0,Y 222.479,Z 249.084,A -85,B 0,C 180,E1 -21029.64,E2 -21029.64} C_VEL
LIN {X 0,Y 221.566,Z 247.159,A -85,B 0,C 180,E1 -21034.142,E2 -21034.142} C_VEL
LIN {X 0,Y 222.045,Z 246.902,A -85,B 0,C 180,E1 -21037.678,E2 -21037.678} C_VEL
LIN {X 0,Y 223.949,Z 248.044,A -85,B 0,C 180,E1 -21041.855,E2 -21041.855} C_VEL
LIN {X 0,Y 225.908,Z 251.026,A -85,B 0,C 180,E1 -21044.666,E2 -21044.666} C_VEL
LIN {X 0,Y 227.713,Z 252.421,A -85,B 0,C 180,E1 -21046.485,E2 -21046.485} C_VEL
LIN {X 0,Y 229.718,Z 255.689,A -85,B 0,C 180,E1 -21048.418,E2 -21048.418} C_VEL
LIN {X 0,Y 231.568,Z 257.695,A -85,B 0,C 180,E1 -21049.839,E2 -21049.839} C_VEL
LIN {X 0,Y 234.915,Z 262.685,A -85,B 0,C 180,E1 -21052.23,E2 -21052.23} C_VEL
LIN {X 0,Y 238.549,Z 267.725,A -85,B 0,C 180,E1 -21054.367,E2 -21054.367} C_VEL
LIN {X 0,Y 241.806,Z 273.159,A -85,B 0,C 180,E1 -21056.147,E2 -21056.147} C_VEL
LIN {X 0,Y 247.953,Z 284.871,A -85,B 0,C 180,E1 -21059.13,E2 -21059.13} C_VEL
LIN {X 0,Y 248.252,Z 285.478,A -85,B 0,C 180,E1 -21059.263,E2 -21059.263} C_VEL
LIN {X 0,Y 244.191,Z 329.909,A -85,B 0,C 180,E1 -21060.885,E2 -21060.885} C_VEL
LIN {X 0,Y 242.495,Z 342.59,A -85,B 0,C 180,E1 -21061.661,E2 -21061.661} C_VEL
LIN {X 0,Y 240.053,Z 355.524,A -85,B 0,C 180,E1 -21062.773,E2 -21062.773} C_VEL
LIN {X 0,Y 237.267,Z 366.614,A -85,B 0,C 180,E1 -21064.034,E2 -21064.034} C_VEL
LIN {X 0,Y 233.736,Z 378.002,A -85,B 0,C 180,E1 -21065.678,E2 -21065.678} C_VEL
LIN {X 0,Y 230.297,Z 387.627,A -85,B 0,C 180,E1 -21067.452,E2 -21067.452} C_VEL
LIN {X 0,Y 226.828,Z 395.98,A -85,B 0,C 180,E1 -21069.361,E2 -21069.361} C_VEL
LIN {X 0,Y 222.692,Z 404.828,A -85,B 0,C 180,E1 -21071.949,E2 -21071.949} C_VEL
LIN {X 0,Y 219.26,Z 411.361,A -85,B 0,C 180,E1 -21074.384,E2 -21074.384} C_VEL
LIN {X 0,Y 216.012,Z 416.957,A -85,B 0,C 180,E1 -21077.027,E2 -21077.027} C_VEL
LIN {X 0,Y 212.74,Z 422.118,A -85,B 0,C 180,E1 -21080.296,E2 -21080.296} C_VEL
LIN {X 0,Y 210.017,Z 425.764,A -85,B 0,C 180,E1 -21083.676,E2 -21083.676} C_VEL
LIN {X 0,Y 208.515,Z 427.461,A -85,B 0,C 180,E1 -21085.987,E2 -21085.987} C_VEL
LIN {X 0,Y 207.241,Z 428.513,A -85,B 0,C 180,E1 -21088.344,E2 -21088.344} C_VEL
LIN {X 0,Y 206.008,Z 429.014,A -85,B 0,C 180,E1 -21091.474,E2 -21091.474} C_VEL
LIN {X 0,Y 205.178,Z 428.451,A -85,B 0,C 180,E1 -21094.707,E2 -21094.707} C_VEL
LIN {X 0,Y 204.763,Z 426.652,A -85,B 0,C 180,E1 -21098.156,E2 -21098.156} C_VEL
LIN {X 0,Y 204.915,Z 423.047,A -85,B 0,C 180,E1 -21102.049,E2 -21102.049} C_VEL
LIN {X 0,Y 205.409,Z 419.312,A -85,B 0,C 180,E1 -21104.875,E2 -21104.875} C_VEL
LIN {X 0,Y 206.071,Z 414.564,A -85,B 0,C 180,E1 -21107.672,E2 -21107.672} C_VEL
LIN {X 0,Y 206.983,Z 408.688,A -85,B 0,C 180,E1 -21110.436,E2 -21110.436} C_VEL
LIN {X 0,Y 208.231,Z 401.109,A -85,B 0,C 180,E1 -21113.301,E2 -21113.301} C_VEL
LIN {X 0,Y 209.878,Z 392.166,A -85,B 0,C 180,E1 -21116.007,E2 -21116.007} C_VEL
LIN {X 0,Y 211.579,Z 382.008,A -85,B 0,C 180,E1 -21118.452,E2 -21118.452} C_VEL
LIN {X 0,Y 213.316,Z 370.919,A -85,B 0,C 180,E1 -21120.591,E2 -21120.591} C_VEL
LIN {X 0,Y 214.81,Z 360.164,A -85,B 0,C 180,E1 -21122.237,E2 -21122.237} C_VEL
LIN {X 0,Y 216.388,Z 346.894,A -85,B 0,C 180,E1 -21123.795,E2 -21123.795} C_VEL
LIN {X 0,Y 217.517,Z 333.78,A -85,B 0,C 180,E1 -21124.924,E2 -21124.924} C_VEL
LIN {X 0,Y 218.305,Z 320.785,A -85,B 0,C 180,E1 -21125.667,E2 -21125.667} C_VEL
LIN {X 0,Y 220.793,Z 263.265,A -85,B 0,C 180,E1 -21127.914,E2 -21127.914} C_VEL
LIN {X 0,Y 212.487,Z 242.534,A -85,B 0,C 180,E1 -21129.711,E2 -21129.711} C_VEL
LIN {X 0,Y 206.988,Z 229.673,A -85,B 0,C 180,E1 -21130.926,E2 -21130.926} C_VEL
LIN {X 0,Y 206.795,Z 228.726,A -85,B 0,C 180,E1 -21131.036,E2 -21131.036} C_VEL
LIN {X 0,Y 206.845,Z 228.72,A -85,B 0,C 180,E1 -21134.228,E2 -21134.228} C_VEL
LIN {X 0,Y 207.062,Z 228.692,A -85,B 0,C 180,E1 -21139.836,E2 -21139.836} C_VEL
LIN {X 0,Y 207.128,Z 228.685,A -85,B 0,C 180,E1 -21142.2,E2 -21142.2} C_VEL
LIN {X 0,Y 207.379,Z 228.652,A -85,B 0,C 180,E1 -21148.058,E2 -21148.058} C_VEL
LIN {X 0,Y 207.509,Z 228.635,A -85,B 0,C 180,E1 -21150.001,E2 -21150.001} C_VEL
LIN {X 0,Y 207.375,Z 228.652,A -85,B 0,C 180,E1 -21151.943,E2 -21151.943} C_VEL
LIN {X 0,Y 207.133,Z 228.682,A -85,B 0,C 180,E1 -21157.801,E2 -21157.801} C_VEL
LIN {X 0,Y 206.927,Z 228.708,A -85,B 0,C 180,E1 -21161.759,E2 -21161.759} C_VEL
LIN {X 0,Y 206.869,Z 228.716,A -85,B 0,C 180,E1 -21165.771,E2 -21165.771} C_VEL
LIN {X 0,Y 206.782,Z 228.72,A -85,B 0,C 180,E1 -21169.87,E2 -21169.87} C_VEL
LIN {X 0,Y 206.74,Z 228.725,A -85,B 0,C 180,E1 -21174.076,E2 -21174.076} C_VEL
LIN {X 0,Y 206.69,Z 228.738,A -85,B 0,C 180,E1 -21178.427,E2 -21178.427} C_VEL
LIN {X 0,Y 206.696,Z 228.732,A -85,B 0,C 180,E1 -21182.959,E2 -21182.959} C_VEL
LIN {X 0,Y 206.669,Z 228.717,A -85,B 0,C 180,E1 -21187.743,E2 -21187.743} C_VEL
LIN {X 0,Y 206.637,Z 228.734,A -85,B 0,C 180,E1 -21191.561,E2 -21191.561} C_VEL
LIN {X 0,Y 206.632,Z 228.746,A -85,B 0,C 180,E1 -21195.583,E2 -21195.583} C_VEL
LIN {X 0,Y 206.652,Z 228.741,A -85,B 0,C 180,E1 -21199.747,E2 -21199.747} C_VEL
LIN {X 0,Y 206.701,Z 228.731,A -85,B 0,C 180,E1 -21204.689,E2 -21204.689} C_VEL
LIN {X 0,Y 206.698,Z 228.738,A -85,B 0,C 180,E1 -21209.335,E2 -21209.335} C_VEL
LIN {X 0,Y 206.707,Z 228.728,A -85,B 0,C 180,E1 -21213.769,E2 -21213.769} C_VEL
LIN {X 0,Y 206.736,Z 228.729,A -85,B 0,C 180,E1 -21218.041,E2 -21218.041} C_VEL
LIN {X 0,Y 206.871,Z 228.713,A -85,B 0,C 180,E1 -21222.196,E2 -21222.196} C_VEL
LIN {X 0,Y 206.882,Z 228.705,A -85,B 0,C 180,E1 -21226.244,E2 -21226.244} C_VEL
LIN {X 0,Y 207.081,Z 228.664,A -85,B 0,C 180,E1 -21230.23,E2 -21230.23} C_VEL
LIN {X 0,Y 207.046,Z 228.682,A -85,B 0,C 180,E1 -21234.155,E2 -21234.155} C_VEL
LIN {X 0,Y 207.376,Z 228.651,A -85,B 0,C 180,E1 -21238.058,E2 -21238.058} C_VEL
LIN {X 0,Y 207.485,Z 228.639,A -85,B 0,C 180,E1 -21240,E2 -21240} C_VEL
LIN {X 0,Y 207.349,Z 228.656,A -85,B 0,C 180,E1 -21241.943,E2 -21241.943} C_VEL
LIN {X 0,Y 207.132,Z 228.667,A -85,B 0,C 180,E1 -21247.8,E2 -21247.8} C_VEL
LIN {X 0,Y 206.917,Z 228.706,A -85,B 0,C 180,E1 -21251.759,E2 -21251.759} C_VEL
LIN {X 0,Y 206.83,Z 228.724,A -85,B 0,C 180,E1 -21255.774,E2 -21255.774} C_VEL
LIN {X 0,Y 206.731,Z 228.727,A -85,B 0,C 180,E1 -21259.875,E2 -21259.875} C_VEL
LIN {X 0,Y 206.724,Z 228.736,A -85,B 0,C 180,E1 -21264.077,E2 -21264.077} C_VEL
LIN {X 0,Y 206.689,Z 228.738,A -85,B 0,C 180,E1 -21268.427,E2 -21268.427} C_VEL
LIN {X 0,Y 206.697,Z 228.736,A -85,B 0,C 180,E1 -21272.958,E2 -21272.958} C_VEL
LIN {X 0,Y 206.671,Z 228.744,A -85,B 0,C 180,E1 -21277.742,E2 -21277.742} C_VEL
LIN {X 0,Y 206.634,Z 228.749,A -85,B 0,C 180,E1 -21281.559,E2 -21281.559} C_VEL
LIN {X 0,Y 206.631,Z 228.747,A -85,B 0,C 180,E1 -21285.583,E2 -21285.583} C_VEL
LIN {X 0,Y 206.71,Z 228.839,A -85,B 0,C 180,E1 -21289.867,E2 -21289.867} C_VEL
LIN {X 0,Y 208.888,Z 238.473,A -85,B 0,C 180,E1 -21293.851,E2 -21293.851} C_VEL
LIN {X 0,Y 210.516,Z 246.187,A -85,B 0,C 180,E1 -21296.845,E2 -21296.845} C_VEL
LIN {X 0,Y 214.889,Z 259.486,A -85,B 0,C 180,E1 -21297.93,E2 -21297.93} C_VEL
LIN {X 0,Y 215.904,Z 270.674,A -85,B 0,C 180,E1 -21298.535,E2 -21298.535} C_VEL
LIN {X 0,Y 215.562,Z 274.632,A -85,B 0,C 180,E1 -21298.677,E2 -21298.677} C_VEL
LIN {X 0,Y 211.32,Z 287.464,A -85,B 0,C 180,E1 -21298.821,E2 -21298.821} C_VEL
LIN {X 0,Y 211.186,Z 291.378,A -85,B 0,C 180,E1 -21298.984,E2 -21298.984} C_VEL
LIN {X 0,Y 212.76,Z 310.455,A -85,B 0,C 180,E1 -21299.997,E2 -21299.997} C_VEL
LIN {X 0,Y 210.563,Z 355.75,A -85,B 0,C 180,E1 -21301.871,E2 -21301.871} C_VEL
LIN {X 0,Y 209.449,Z 369.23,A -85,B 0,C 180,E1 -21302.794,E2 -21302.794} C_VEL
LIN {X 0,Y 207.983,Z 381.095,A -85,B 0,C 180,E1 -21303.941,E2 -21303.941} C_VEL
LIN {X 0,Y 206.091,Z 393.573,A -85,B 0,C 180,E1 -21305.576,E2 -21305.576} C_VEL
LIN {X 0,Y 204.203,Z 404.829,A -85,B 0,C 180,E1 -21307.487,E2 -21307.487} C_VEL
LIN {X 0,Y 202.354,Z 415.03,A -85,B 0,C 180,E1 -21309.676,E2 -21309.676} C_VEL
LIN {X 0,Y 200.648,Z 424.239,A -85,B 0,C 180,E1 -21312.152,E2 -21312.152} C_VEL
LIN {X 0,Y 199.334,Z 433.261,A -85,B 0,C 180,E1 -21315.189,E2 -21315.189} C_VEL
LIN {X 0,Y 198.33,Z 440.388,A -85,B 0,C 180,E1 -21318.243,E2 -21318.243} C_VEL
LIN {X 0,Y 197.964,Z 445.229,A -85,B 0,C 180,E1 -21320.807,E2 -21320.807} C_VEL
LIN {X 0,Y 197.964,Z 450.635,A -85,B 0,C 180,E1 -21324.554,E2 -21324.554} C_VEL
LIN {X 0,Y 197.979,Z 454.056,A -85,B 0,C 180,E1 -21327.965,E2 -21327.965} C_VEL
LIN {X 0,Y 198.297,Z 455.505,A -85,B 0,C 180,E1 -21329.999,E2 -21329.999} C_VEL
LIN {X 0,Y 197.686,Z 456.873,A -85,B 0,C 180,E1 -21334.077,E2 -21334.077} C_VEL
LIN {X 0,Y 197.558,Z 456.652,A -85,B 0,C 180,E1 -21338.18,E2 -21338.18} C_VEL
LIN {X 0,Y 198.315,Z 454.818,A -85,B 0,C 180,E1 -21342.276,E2 -21342.276} C_VEL
LIN {X 0,Y 199.025,Z 453.32,A -85,B 0,C 180,E1 -21344.31,E2 -21344.31} C_VEL
LIN {X 0,Y 200.817,Z 450.308,A -85,B 0,C 180,E1 -21347.305,E2 -21347.305} C_VEL
LIN {X 0,Y 203.068,Z 446.304,A -85,B 0,C 180,E1 -21350.248,E2 -21350.248} C_VEL
LIN {X 0,Y 205.739,Z 441.24,A -85,B 0,C 180,E1 -21353.131,E2 -21353.131} C_VEL
LIN {X 0,Y 209.853,Z 433.842,A -85,B 0,C 180,E1 -21356.343,E2 -21356.343} C_VEL
LIN {X 0,Y 214.035,Z 425.909,A -85,B 0,C 180,E1 -21358.968,E2 -21358.968} C_VEL
LIN {X 0,Y 218.674,Z 416.13,A -85,B 0,C 180,E1 -21361.484,E2 -21361.484} C_VEL
LIN {X 0,Y 222.998,Z 406.184,A -85,B 0,C 180,E1 -21363.471,E2 -21363.471} C_VEL
LIN {X 0,Y 227.194,Z 395.258,A -85,B 0,C 180,E1 -21365.179,E2 -21365.179} C_VEL
LIN {X 0,Y 231.23,Z 383.101,A -85,B 0,C 180,E1 -21366.618,E2 -21366.618} C_VEL
LIN {X 0,Y 234.684,Z 370.385,A -85,B 0,C 180,E1 -21367.736,E2 -21367.736} C_VEL
LIN {X 0,Y 237.484,Z 356.361,A -85,B 0,C 180,E1 -21368.62,E2 -21368.62} C_VEL
LIN {X 0,Y 239.229,Z 342.345,A -85,B 0,C 180,E1 -21369.229,E2 -21369.229} C_VEL
LIN {X 0,Y 241.635,Z 315.736,A -85,B 0,C 180,E1 -21370.199,E2 -21370.199} C_VEL
LIN {X 0,Y 241.249,Z 302.816,A -85,B 0,C 180,E1 -21371.226,E2 -21371.226} C_VEL
LIN {X 0,Y 240.854,Z 296.954,A -85,B 0,C 180,E1 -21371.785,E2 -21371.785} C_VEL
LIN {X 0,Y 237.572,Z 288.143,A -85,B 0,C 180,E1 -21373.691,E2 -21373.691} C_VEL
LIN {X 0,Y 234.679,Z 281.635,A -85,B 0,C 180,E1 -21375.508,E2 -21375.508} C_VEL
LIN {X 0,Y 231.009,Z 273.98,A -85,B 0,C 180,E1 -21378.081,E2 -21378.081} C_VEL
LIN {X 0,Y 227.618,Z 267.5,A -85,B 0,C 180,E1 -21380.891,E2 -21380.891} C_VEL
LIN {X 0,Y 224.273,Z 261.32,A -85,B 0,C 180,E1 -21384.498,E2 -21384.498} C_VEL
LIN {X 0,Y 221.167,Z 255.925,A -85,B 0,C 180,E1 -21389.968,E2 -21389.968} C_VEL
LIN {X 0,Y 220.379,Z 254.079,A -85,B 0,C 180,E1 -21394.499,E2 -21394.499} C_VEL
LIN {X 0,Y 221.113,Z 254.063,A -85,B 0,C 180,E1 -21398.56,E2 -21398.56} C_VEL
LIN {X 0,Y 222.637,Z 255.136,A -85,B 0,C 180,E1 -21401.699,E2 -21401.699} C_VEL
LIN {X 0,Y 224.54,Z 257.976,A -85,B 0,C 180,E1 -21404.501,E2 -21404.501} C_VEL
LIN {X 0,Y 226.011,Z 259.297,A -85,B 0,C 180,E1 -21406.089,E2 -21406.089} C_VEL
LIN {X 0,Y 228.339,Z 262.811,A -85,B 0,C 180,E1 -21408.347,E2 -21408.347} C_VEL
LIN {X 0,Y 229.583,Z 264.303,A -85,B 0,C 180,E1 -21409.365,E2 -21409.365} C_VEL
LIN {X 0,Y 232.682,Z 269.092,A -85,B 0,C 180,E1 -21411.668,E2 -21411.668} C_VEL
LIN {X 0,Y 236.042,Z 273.946,A -85,B 0,C 180,E1 -21413.771,E2 -21413.771} C_VEL
LIN {X 0,Y 238.953,Z 279.01,A -85,B 0,C 180,E1 -21415.471,E2 -21415.471} C_VEL
LIN {X 0,Y 243.851,Z 288.844,A -85,B 0,C 180,E1 -21418.027,E2 -21418.027} C_VEL
LIN {X 0,Y 239.776,Z 330.667,A -85,B 0,C 180,E1 -21419.581,E2 -21419.581} C_VEL
LIN {X 0,Y 237.881,Z 344.091,A -85,B 0,C 180,E1 -21420.423,E2 -21420.423} C_VEL
LIN {X 0,Y 235.406,Z 356.38,A -85,B 0,C 180,E1 -21421.497,E2 -21421.497} C_VEL
LIN {X 0,Y 232.218,Z 368.349,A -85,B 0,C 180,E1 -21422.889,E2 -21422.889} C_VEL
LIN {X 0,Y 228.811,Z 378.642,A -85,B 0,C 180,E1 -21424.404,E2 -21424.404} C_VEL
LIN {X 0,Y 224.863,Z 388.953,A -85,B 0,C 180,E1 -21426.351,E2 -21426.351} C_VEL
LIN {X 0,Y 220.425,Z 398.79,A -85,B 0,C 180,E1 -21428.737,E2 -21428.737} C_VEL
LIN {X 0,Y 216.396,Z 406.818,A -85,B 0,C 180,E1 -21431.237,E2 -21431.237} C_VEL
LIN {X 0,Y 213.331,Z 412.192,A -85,B 0,C 180,E1 -21433.333,E2 -21433.333} C_VEL
LIN {X 0,Y 210.538,Z 416.711,A -85,B 0,C 180,E1 -21435.489,E2 -21435.489} C_VEL
LIN {X 0,Y 207.336,Z 421.421,A -85,B 0,C 180,E1 -21438.36,E2 -21438.36} C_VEL
LIN {X 0,Y 204.278,Z 425.421,A -85,B 0,C 180,E1 -21441.735,E2 -21441.735} C_VEL
LIN {X 0,Y 201.869,Z 428.042,A -85,B 0,C 180,E1 -21445.154,E2 -21445.154} C_VEL
LIN {X 0,Y 200.039,Z 429.371,A -85,B 0,C 180,E1 -21448.56,E2 -21448.56} C_VEL
LIN {X 0,Y 198.732,Z 429.518,A -85,B 0,C 180,E1 -21452.037,E2 -21452.037} C_VEL
LIN {X 0,Y 198.004,Z 428.608,A -85,B 0,C 180,E1 -21455.278,E2 -21455.278} C_VEL
LIN {X 0,Y 197.655,Z 426.66,A -85,B 0,C 180,E1 -21458.533,E2 -21458.533} C_VEL
LIN {X 0,Y 197.871,Z 422.879,A -85,B 0,C 180,E1 -21462.442,E2 -21462.442} C_VEL
LIN {X 0,Y 198.487,Z 418.246,A -85,B 0,C 180,E1 -21465.808,E2 -21465.808} C_VEL
LIN {X 0,Y 199.435,Z 411.914,A -85,B 0,C 180,E1 -21469.258,E2 -21469.258} C_VEL
LIN {X 0,Y 200.748,Z 404.352,A -85,B 0,C 180,E1 -21472.472,E2 -21472.472} C_VEL
LIN {X 0,Y 202.18,Z 396.329,A -85,B 0,C 180,E1 -21475.194,E2 -21475.194} C_VEL
LIN {X 0,Y 203.787,Z 387.226,A -85,B 0,C 180,E1 -21477.687,E2 -21477.687} C_VEL
LIN {X 0,Y 205.582,Z 376.696,A -85,B 0,C 180,E1 -21480.015,E2 -21480.015} C_VEL
LIN {X 0,Y 207.289,Z 365.31,A -85,B 0,C 180,E1 -21482.016,E2 -21482.016} C_VEL
LIN {X 0,Y 208.906,Z 353.218,A -85,B 0,C 180,E1 -21483.663,E2 -21483.663} C_VEL
LIN {X 0,Y 210.186,Z 341.165,A -85,B 0,C 180,E1 -21484.919,E2 -21484.919} C_VEL
LIN {X 0,Y 211.106,Z 328.039,A -85,B 0,C 180,E1 -21485.9,E2 -21485.9} C_VEL
LIN {X 0,Y 211.937,Z 310.944,A -85,B 0,C 180,E1 -21486.69,E2 -21486.69} C_VEL
LIN {X 0,Y 214.202,Z 265.002,A -85,B 0,C 180,E1 -21488.515,E2 -21488.515} C_VEL
LIN {X 0,Y 204.469,Z 241.033,A -85,B 0,C 180,E1 -21490.681,E2 -21490.681} C_VEL
LIN {X 0,Y 199.968,Z 230.47,A -85,B 0,C 180,E1 -21491.74,E2 -21491.74} C_VEL
LIN {X 0,Y 199.812,Z 229.595,A -85,B 0,C 180,E1 -21491.845,E2 -21491.845} C_VEL
LIN {X 0,Y 199.82,Z 229.594,A -85,B 0,C 180,E1 -21495.748,E2 -21495.748} C_VEL
LIN {X 0,Y 200.023,Z 229.569,A -85,B 0,C 180,E1 -21499.882,E2 -21499.882} C_VEL
LIN {X 0,Y 200.011,Z 229.57,A -85,B 0,C 180,E1 -21503.95,E2 -21503.95} C_VEL
LIN {X 0,Y 200.318,Z 229.531,A -85,B 0,C 180,E1 -21507.99,E2 -21507.99} C_VEL
LIN {X 0,Y 200.474,Z 229.512,A -85,B 0,C 180,E1 -21510.001,E2 -21510.001} C_VEL
LIN {X 0,Y 200.012,Z 229.57,A -85,B 0,C 180,E1 -21514.03,E2 -21514.03} C_VEL
LIN {X 0,Y 200.083,Z 229.561,A -85,B 0,C 180,E1 -21518.077,E2 -21518.077} C_VEL
LIN {X 0,Y 199.877,Z 229.588,A -85,B 0,C 180,E1 -21522.18,E2 -21522.18} C_VEL
LIN {X 0,Y 199.807,Z 229.596,A -85,B 0,C 180,E1 -21526.344,E2 -21526.344} C_VEL
LIN {X 0,Y 199.693,Z 229.598,A -85,B 0,C 180,E1 -21530.607,E2 -21530.607} C_VEL
LIN {X 0,Y 199.653,Z 229.609,A -85,B 0,C 180,E1 -21534.988,E2 -21534.988} C_VEL
LIN {X 0,Y 199.61,Z 229.621,A -85,B 0,C 180,E1 -21539.533,E2 -21539.533} C_VEL
LIN {X 0,Y 199.667,Z 229.608,A -85,B 0,C 180,E1 -21542.353,E2 -21542.353} C_VEL
LIN {X 0,Y 199.619,Z 229.598,A -85,B 0,C 180,E1 -21546.765,E2 -21546.765} C_VEL
LIN {X 0,Y 199.597,Z 229.6,A -85,B 0,C 180,E1 -21549.332,E2 -21549.332} C_VEL
LIN {X 0,Y 199.571,Z 229.616,A -85,B 0,C 180,E1 -21552.309,E2 -21552.309} C_VEL
LIN {X 0,Y 199.578,Z 229.622,A -85,B 0,C 180,E1 -21555.228,E2 -21555.228} C_VEL
LIN {X 0,Y 199.575,Z 229.624,A -85,B 0,C 180,E1 -21558.004,E2 -21558.004} C_VEL
LIN {X 0,Y 199.602,Z 229.619,A -85,B 0,C 180,E1 -21560.772,E2 -21560.772} C_VEL
LIN {X 0,Y 199.615,Z 229.613,A -85,B 0,C 180,E1 -21564.075,E2 -21564.075} C_VEL
LIN {X 0,Y 199.688,Z 229.609,A -85,B 0,C 180,E1 -21568.135,E2 -21568.135} C_VEL
LIN {X 0,Y 199.646,Z 229.613,A -85,B 0,C 180,E1 -21572.766,E2 -21572.766} C_VEL
LIN {X 0,Y 199.71,Z 229.606,A -85,B 0,C 180,E1 -21577.226,E2 -21577.226} C_VEL
LIN {X 0,Y 199.798,Z 229.594,A -85,B 0,C 180,E1 -21581.759,E2 -21581.759} C_VEL
LIN {X 0,Y 199.822,Z 229.583,A -85,B 0,C 180,E1 -21585.747,E2 -21585.747} C_VEL
LIN {X 0,Y 200.026,Z 229.541,A -85,B 0,C 180,E1 -21589.882,E2 -21589.882} C_VEL
LIN {X 0,Y 200.009,Z 229.557,A -85,B 0,C 180,E1 -21593.949,E2 -21593.949} C_VEL
LIN {X 0,Y 200.315,Z 229.53,A -85,B 0,C 180,E1 -21597.99,E2 -21597.99} C_VEL
LIN {X 0,Y 200.452,Z 229.515,A -85,B 0,C 180,E1 -21600,E2 -21600} C_VEL
LIN {X 0,Y 199.995,Z 229.569,A -85,B 0,C 180,E1 -21604.03,E2 -21604.03} C_VEL
LIN {X 0,Y 200.08,Z 229.545,A -85,B 0,C 180,E1 -21608.077,E2 -21608.077} C_VEL
LIN {X 0,Y 199.867,Z 229.586,A -85,B 0,C 180,E1 -21612.18,E2 -21612.18} C_VEL
LIN {X 0,Y 199.767,Z 229.602,A -85,B 0,C 180,E1 -21616.347,E2 -21616.347} C_VEL
LIN {X 0,Y 199.66,Z 229.604,A -85,B 0,C 180,E1 -21620.61,E2 -21620.61} C_VEL
LIN {X 0,Y 199.639,Z 229.617,A -85,B 0,C 180,E1 -21624.989,E2 -21624.989} C_VEL
LIN {X 0,Y 199.61,Z 229.618,A -85,B 0,C 180,E1 -21629.533,E2 -21629.533} C_VEL
LIN {X 0,Y 199.668,Z 229.611,A -85,B 0,C 180,E1 -21632.352,E2 -21632.352} C_VEL
LIN {X 0,Y 199.62,Z 229.618,A -85,B 0,C 180,E1 -21636.764,E2 -21636.764} C_VEL
LIN {X 0,Y 199.597,Z 229.625,A -85,B 0,C 180,E1 -21639.331,E2 -21639.331} C_VEL
LIN {X 0,Y 199.568,Z 229.627,A -85,B 0,C 180,E1 -21642.307,E2 -21642.307} C_VEL
LIN {X 0,Y 199.578,Z 229.626,A -85,B 0,C 180,E1 -21645.227,E2 -21645.227} C_VEL
LIN {X 0,Y 199.613,Z 229.624,A -85,B 0,C 180,E1 -21649.274,E2 -21649.274} C_VEL
LIN {X 0,Y 201.733,Z 238.899,A -85,B 0,C 180,E1 -21653.253,E2 -21653.253} C_VEL
LIN {X 0,Y 203.103,Z 245.457,A -85,B 0,C 180,E1 -21655.946,E2 -21655.946} C_VEL
LIN {X 0,Y 208.371,Z 261.231,A -85,B 0,C 180,E1 -21657.302,E2 -21657.302} C_VEL
LIN {X 0,Y 211.186,Z 291.378,A -85,B 0,C 180,E1 -21658.984,E2 -21658.984} C_VEL
LIN {X 0,Y 211.355,Z 295.257,A -85,B 0,C 180,E1 -21659.176,E2 -21659.176} C_VEL
LIN {X 0,Y 210.899,Z 299.144,A -85,B 0,C 180,E1 -21659.306,E2 -21659.306} C_VEL
LIN {X 0,Y 208.892,Z 306.858,A -85,B 0,C 180,E1 -21659.458,E2 -21659.458} C_VEL
LIN {X 0,Y 206.133,Z 316.566,A -85,B 0,C 180,E1 -21659.638,E2 -21659.638} C_VEL
LIN {X 0,Y 205.443,Z 322.5,A -85,B 0,C 180,E1 -21659.849,E2 -21659.849} C_VEL
LIN {X 0,Y 203.718,Z 356.264,A -85,B 0,C 180,E1 -21661.331,E2 -21661.331} C_VEL
LIN {X 0,Y 202.681,Z 368.723,A -85,B 0,C 180,E1 -21662.228,E2 -21662.228} C_VEL
LIN {X 0,Y 201.031,Z 381.552,A -85,B 0,C 180,E1 -21663.529,E2 -21663.529} C_VEL
LIN {X 0,Y 199.101,Z 393.789,A -85,B 0,C 180,E1 -21665.217,E2 -21665.217} C_VEL
LIN {X 0,Y 197.176,Z 404.895,A -85,B 0,C 180,E1 -21667.193,E2 -21667.193} C_VEL
LIN {X 0,Y 195.236,Z 415.206,A -85,B 0,C 180,E1 -21669.526,E2 -21669.526} C_VEL
LIN {X 0,Y 193.571,Z 424.069,A -85,B 0,C 180,E1 -21672.024,E2 -21672.024} C_VEL
LIN {X 0,Y 192.221,Z 433.021,A -85,B 0,C 180,E1 -21675.17,E2 -21675.17} C_VEL
LIN {X 0,Y 191.228,Z 440.079,A -85,B 0,C 180,E1 -21678.337,E2 -21678.337} C_VEL
LIN {X 0,Y 190.868,Z 445.704,A -85,B 0,C 180,E1 -21681.53,E2 -21681.53} C_VEL
LIN {X 0,Y 190.917,Z 449.8,A -85,B 0,C 180,E1 -21684.511,E2 -21684.511} C_VEL
LIN {X 0,Y 190.911,Z 453.172,A -85,B 0,C 180,E1 -21687.89,E2 -21687.89} C_VEL
LIN {X 0,Y 191.237,Z 454.697,A -85,B 0,C 180,E1 -21689.999,E2 -21689.999} C_VEL
LIN {X 0,Y 190.767,Z 455.685,A -85,B 0,C 180,E1 -21692.111,E2 -21692.111} C_VEL
LIN {X 0,Y 190.492,Z 456.337,A -85,B 0,C 180,E1 -21695.036,E2 -21695.036} C_VEL
LIN {X 0,Y 190.498,Z 456.142,A -85,B 0,C 180,E1 -21698.486,E2 -21698.486} C_VEL
LIN {X 0,Y 190.809,Z 455.526,A -85,B 0,C 180,E1 -21700.612,E2 -21700.612} C_VEL
LIN {X 0,Y 191.325,Z 454.509,A -85,B 0,C 180,E1 -21702.732,E2 -21702.732} C_VEL
LIN {X 0,Y 192.128,Z 453.081,A -85,B 0,C 180,E1 -21704.836,E2 -21704.836} C_VEL
LIN {X 0,Y 194.698,Z 449.043,A -85,B 0,C 180,E1 -21708.957,E2 -21708.957} C_VEL
LIN {X 0,Y 197.538,Z 444.329,A -85,B 0,C 180,E1 -21712.327,E2 -21712.327} C_VEL
LIN {X 0,Y 200.965,Z 438.652,A -85,B 0,C 180,E1 -21715.365,E2 -21715.365} C_VEL
LIN {X 0,Y 204.942,Z 431.923,A -85,B 0,C 180,E1 -21718.133,E2 -21718.133} C_VEL
LIN {X 0,Y 210.214,Z 422.207,A -85,B 0,C 180,E1 -21721.211,E2 -21721.211} C_VEL
LIN {X 0,Y 214.46,Z 413.687,A -85,B 0,C 180,E1 -21723.292,E2 -21723.292} C_VEL
LIN {X 0,Y 219.107,Z 403.323,A -85,B 0,C 180,E1 -21725.265,E2 -21725.265} C_VEL
LIN {X 0,Y 223.592,Z 391.864,A -85,B 0,C 180,E1 -21726.951,E2 -21726.951} C_VEL
LIN {X 0,Y 227.324,Z 380.754,A -85,B 0,C 180,E1 -21728.193,E2 -21728.193} C_VEL
LIN {X 0,Y 230.869,Z 367.419,A -85,B 0,C 180,E1 -21729.313,E2 -21729.313} C_VEL
LIN {X 0,Y 233.574,Z 353.901,A -85,B 0,C 180,E1 -21730.13,E2 -21730.13} C_VEL
LIN {X 0,Y 235.622,Z 336.651,A -85,B 0,C 180,E1 -21730.825,E2 -21730.825} C_VEL
LIN {X 0,Y 237.516,Z 316.827,A -85,B 0,C 180,E1 -21731.566,E2 -21731.566} C_VEL
LIN {X 0,Y 237.205,Z 303.324,A -85,B 0,C 180,E1 -21732.681,E2 -21732.681} C_VEL
LIN {X 0,Y 237.019,Z 300.564,A -85,B 0,C 180,E1 -21732.958,E2 -21732.958} C_VEL
LIN {X 0,Y 234.161,Z 292.558,A -85,B 0,C 180,E1 -21734.804,E2 -21734.804} C_VEL
LIN {X 0,Y 230.883,Z 284.936,A -85,B 0,C 180,E1 -21737.043,E2 -21737.043} C_VEL
LIN {X 0,Y 228.277,Z 279.388,A -85,B 0,C 180,E1 -21739.091,E2 -21739.091} C_VEL
LIN {X 0,Y 225.432,Z 273.545,A -85,B 0,C 180,E1 -21741.702,E2 -21741.702} C_VEL
LIN {X 0,Y 222.539,Z 267.856,A -85,B 0,C 180,E1 -21745.112,E2 -21745.112} C_VEL
LIN {X 0,Y 219.891,Z 262.884,A -85,B 0,C 180,E1 -21750.172,E2 -21750.172} C_VEL
LIN {X 0,Y 219.198,Z 261.044,A -85,B 0,C 180,E1 -21754.606,E2 -21754.606} C_VEL
LIN {X 0,Y 219.769,Z 260.964,A -85,B 0,C 180,E1 -21758.031,E2 -21758.031} C_VEL
LIN {X 0,Y 221.228,Z 261.996,A -85,B 0,C 180,E1 -21761.344,E2 -21761.344} C_VEL
LIN {X 0,Y 223.223,Z 264.974,A -85,B 0,C 180,E1 -21764.407,E2 -21764.407} C_VEL
LIN {X 0,Y 224.335,Z 266.118,A -85,B 0,C 180,E1 -21765.703,E2 -21765.703} C_VEL
LIN {X 0,Y 226.765,Z 269.663,A -85,B 0,C 180,E1 -21768.097,E2 -21768.097} C_VEL
LIN {X 0,Y 227.88,Z 271.354,A -85,B 0,C 180,E1 -21769.099,E2 -21769.099} C_VEL
LIN {X 0,Y 230.451,Z 275.396,A -85,B 0,C 180,E1 -21771.073,E2 -21771.073} C_VEL
LIN {X 0,Y 233.711,Z 280.326,A -85,B 0,C 180,E1 -21773.25,E2 -21773.25} C_VEL
LIN {X 0,Y 236.643,Z 285.84,A -85,B 0,C 180,E1 -21775.044,E2 -21775.044} C_VEL
LIN {X 0,Y 239.646,Z 292.081,A -85,B 0,C 180,E1 -21776.733,E2 -21776.733} C_VEL
LIN {X 0,Y 235.905,Z 329.28,A -85,B 0,C 180,E1 -21778.114,E2 -21778.114} C_VEL
LIN {X 0,Y 234.028,Z 342.321,A -85,B 0,C 180,E1 -21778.866,E2 -21778.866} C_VEL
LIN {X 0,Y 231.336,Z 355.574,A -85,B 0,C 180,E1 -21780,E2 -21780} C_VEL
LIN {X 0,Y 228.112,Z 367.344,A -85,B 0,C 180,E1 -21781.324,E2 -21781.324} C_VEL
LIN {X 0,Y 224.323,Z 378.558,A -85,B 0,C 180,E1 -21782.955,E2 -21782.955} C_VEL
LIN {X 0,Y 220.168,Z 388.997,A -85,B 0,C 180,E1 -21784.906,E2 -21784.906} C_VEL
LIN {X 0,Y 216.012,Z 397.845,A -85,B 0,C 180,E1 -21787.008,E2 -21787.008} C_VEL
LIN {X 0,Y 211.575,Z 406.202,A -85,B 0,C 180,E1 -21789.56,E2 -21789.56} C_VEL
LIN {X 0,Y 207.496,Z 413.011,A -85,B 0,C 180,E1 -21792.22,E2 -21792.22} C_VEL
LIN {X 0,Y 203.772,Z 418.623,A -85,B 0,C 180,E1 -21795.05,E2 -21795.05} C_VEL
LIN {X 0,Y 200.031,Z 423.569,A -85,B 0,C 180,E1 -21798.446,E2 -21798.446} C_VEL
LIN {X 0,Y 196.95,Z 427.028,A -85,B 0,C 180,E1 -21801.908,E2 -21801.908} C_VEL
LIN {X 0,Y 194.37,Z 429.312,A -85,B 0,C 180,E1 -21805.715,E2 -21805.715} C_VEL
LIN {X 0,Y 192.744,Z 430.123,A -85,B 0,C 180,E1 -21808.943,E2 -21808.943} C_VEL
LIN {X 0,Y 191.509,Z 429.926,A -85,B 0,C 180,E1 -21812.43,E2 -21812.43} C_VEL
LIN {X 0,Y 190.774,Z 428.522,A -85,B 0,C 180,E1 -21816.117,E2 -21816.117} C_VEL
LIN {X 0,Y 190.606,Z 425.369,A -85,B 0,C 180,E1 -21820.323,E2 -21820.323} C_VEL
LIN {X 0,Y 190.925,Z 422.023,A -85,B 0,C 180,E1 -21823.36,E2 -21823.36} C_VEL
LIN {X 0,Y 191.727,Z 416.427,A -85,B 0,C 180,E1 -21827.149,E2 -21827.149} C_VEL
LIN {X 0,Y 192.732,Z 409.92,A -85,B 0,C 180,E1 -21830.48,E2 -21830.48} C_VEL
LIN {X 0,Y 194.165,Z 401.64,A -85,B 0,C 180,E1 -21833.814,E2 -21833.814} C_VEL
LIN {X 0,Y 195.903,Z 392.617,A -85,B 0,C 180,E1 -21836.69,E2 -21836.69} C_VEL
LIN {X 0,Y 197.699,Z 382.47,A -85,B 0,C 180,E1 -21839.273,E2 -21839.273} C_VEL
LIN {X 0,Y 199.457,Z 372.035,A -85,B 0,C 180,E1 -21841.408,E2 -21841.408} C_VEL
LIN {X 0,Y 201.262,Z 359.799,A -85,B 0,C 180,E1 -21843.373,E2 -21843.373} C_VEL
LIN {X 0,Y 202.748,Z 347.854,A -85,B 0,C 180,E1 -21844.848,E2 -21844.848} C_VEL
LIN {X 0,Y 203.947,Z 334.906,A -85,B 0,C 180,E1 -21846.037,E2 -21846.037} C_VEL
LIN {X 0,Y 204.758,Z 322.139,A -85,B 0,C 180,E1 -21846.825,E2 -21846.825} C_VEL
LIN {X 0,Y 207.401,Z 266.283,A -85,B 0,C 180,E1 -21849.161,E2 -21849.161} C_VEL
LIN {X 0,Y 197.605,Z 242.26,A -85,B 0,C 180,E1 -21851.453,E2 -21851.453} C_VEL
LIN {X 0,Y 192.865,Z 231.042,A -85,B 0,C 180,E1 -21852.625,E2 -21852.625} C_VEL
LIN {X 0,Y 192.778,Z 230.472,A -85,B 0,C 180,E1 -21852.703,E2 -21852.703} C_VEL
LIN {X 0,Y 192.794,Z 230.47,A -85,B 0,C 180,E1 -21857.367,E2 -21857.367} C_VEL
LIN {X 0,Y 193.026,Z 230.44,A -85,B 0,C 180,E1 -21861.626,E2 -21861.626} C_VEL
LIN {X 0,Y 193.26,Z 230.41,A -85,B 0,C 180,E1 -21867.917,E2 -21867.917} C_VEL
LIN {X 0,Y 193.438,Z 230.388,A -85,B 0,C 180,E1 -21870.001,E2 -21870.001} C_VEL
LIN {X 0,Y 192.958,Z 230.449,A -85,B 0,C 180,E1 -21874.178,E2 -21874.178} C_VEL
LIN {X 0,Y 193.032,Z 230.44,A -85,B 0,C 180,E1 -21878.375,E2 -21878.375} C_VEL
LIN {X 0,Y 192.804,Z 230.468,A -85,B 0,C 180,E1 -21882.634,E2 -21882.634} C_VEL
LIN {X 0,Y 192.76,Z 230.472,A -85,B 0,C 180,E1 -21886.959,E2 -21886.959} C_VEL
LIN {X 0,Y 192.622,Z 230.477,A -85,B 0,C 180,E1 -21891.4,E2 -21891.4} C_VEL
LIN {X 0,Y 192.641,Z 230.481,A -85,B 0,C 180,E1 -21894.209,E2 -21894.209} C_VEL
LIN {X 0,Y 192.604,Z 230.492,A -85,B 0,C 180,E1 -21898.867,E2 -21898.867} C_VEL
LIN {X 0,Y 192.596,Z 230.489,A -85,B 0,C 180,E1 -21903.187,E2 -21903.187} C_VEL
LIN {X 0,Y 192.543,Z 230.475,A -85,B 0,C 180,E1 -21908.355,E2 -21908.355} C_VEL
LIN {X 0,Y 192.489,Z 230.499,A -85,B 0,C 180,E1 -21913.095,E2 -21913.095} C_VEL
LIN {X 0,Y 192.489,Z 230.507,A -85,B 0,C 180,E1 -21916.906,E2 -21916.906} C_VEL
LIN {X 0,Y 192.546,Z 230.494,A -85,B 0,C 180,E1 -21921.647,E2 -21921.647} C_VEL
LIN {X 0,Y 192.597,Z 230.492,A -85,B 0,C 180,E1 -21926.814,E2 -21926.814} C_VEL
LIN {X 0,Y 192.623,Z 230.487,A -85,B 0,C 180,E1 -21931.685,E2 -21931.685} C_VEL
LIN {X 0,Y 192.681,Z 230.477,A -85,B 0,C 180,E1 -21936.345,E2 -21936.345} C_VEL
LIN {X 0,Y 192.733,Z 230.474,A -85,B 0,C 180,E1 -21941.46,E2 -21941.46} C_VEL
LIN {X 0,Y 192.751,Z 230.464,A -85,B 0,C 180,E1 -21945.213,E2 -21945.213} C_VEL
LIN {X 0,Y 192.948,Z 230.421,A -85,B 0,C 180,E1 -21949.567,E2 -21949.567} C_VEL
LIN {X 0,Y 192.972,Z 230.432,A -85,B 0,C 180,E1 -21953.728,E2 -21953.728} C_VEL
LIN {X 0,Y 193.257,Z 230.409,A -85,B 0,C 180,E1 -21957.916,E2 -21957.916} C_VEL
LIN {X 0,Y 193.419,Z 230.392,A -85,B 0,C 180,E1 -21960,E2 -21960} C_VEL
LIN {X 0,Y 192.942,Z 230.445,A -85,B 0,C 180,E1 -21964.178,E2 -21964.178} C_VEL
LIN {X 0,Y 193.03,Z 230.422,A -85,B 0,C 180,E1 -21968.374,E2 -21968.374} C_VEL
LIN {X 0,Y 192.793,Z 230.469,A -85,B 0,C 180,E1 -21972.634,E2 -21972.634} C_VEL
LIN {X 0,Y 192.721,Z 230.478,A -85,B 0,C 180,E1 -21976.962,E2 -21976.962} C_VEL
LIN {X 0,Y 192.589,Z 230.484,A -85,B 0,C 180,E1 -21981.403,E2 -21981.403} C_VEL
LIN {X 0,Y 192.63,Z 230.492,A -85,B 0,C 180,E1 -21984.199,E2 -21984.199} C_VEL
LIN {X 0,Y 192.603,Z 230.492,A -85,B 0,C 180,E1 -21988.865,E2 -21988.865} C_VEL
LIN {X 0,Y 192.597,Z 230.493,A -85,B 0,C 180,E1 -21993.186,E2 -21993.186} C_VEL
LIN {X 0,Y 192.544,Z 230.502,A -85,B 0,C 180,E1 -21998.354,E2 -21998.354} C_VEL
LIN {X 0,Y 192.487,Z 230.511,A -85,B 0,C 180,E1 -22003.093,E2 -22003.093} C_VEL
LIN {X 0,Y 192.575,Z 230.499,A -85,B 0,C 180,E1 -22008.695,E2 -22008.695} C_VEL
LIN {X 0,Y 194.849,Z 240.624,A -85,B 0,C 180,E1 -22013.194,E2 -22013.194} C_VEL
LIN {X 0,Y 195.739,Z 244.899,A -85,B 0,C 180,E1 -22015.013,E2 -22015.013} C_VEL
LIN {X 0,Y 201.868,Z 263.302,A -85,B 0,C 180,E1 -22016.674,E2 -22016.674} C_VEL
LIN {X 0,Y 206.074,Z 310.221,A -85,B 0,C 180,E1 -22019.339,E2 -22019.339} C_VEL
LIN {X 0,Y 205.443,Z 322.5,A -85,B 0,C 180,E1 -22019.849,E2 -22019.849} C_VEL
LIN {X 0,Y 204.674,Z 328.308,A -85,B 0,C 180,E1 -22020.044,E2 -22020.044} C_VEL
LIN {X 0,Y 201.456,Z 337.689,A -85,B 0,C 180,E1 -22020.178,E2 -22020.178} C_VEL
LIN {X 0,Y 198.107,Z 347.057,A -85,B 0,C 180,E1 -22020.324,E2 -22020.324} C_VEL
LIN {X 0,Y 197.155,Z 352.854,A -85,B 0,C 180,E1 -22020.546,E2 -22020.546} C_VEL
LIN {X 0,Y 196.151,Z 365.847,A -85,B 0,C 180,E1 -22021.438,E2 -22021.438} C_VEL
LIN {X 0,Y 194.519,Z 378.765,A -85,B 0,C 180,E1 -22022.715,E2 -22022.715} C_VEL
LIN {X 0,Y 192.631,Z 390.788,A -85,B 0,C 180,E1 -22024.325,E2 -22024.325} C_VEL
LIN {X 0,Y 190.615,Z 402.33,A -85,B 0,C 180,E1 -22026.361,E2 -22026.361} C_VEL
LIN {X 0,Y 188.723,Z 412.359,A -85,B 0,C 180,E1 -22028.591,E2 -22028.591} C_VEL
LIN {X 0,Y 186.771,Z 422.234,A -85,B 0,C 180,E1 -22031.346,E2 -22031.346} C_VEL
LIN {X 0,Y 185.51,Z 430.022,A -85,B 0,C 180,E1 -22034.057,E2 -22034.057} C_VEL
LIN {X 0,Y 184.405,Z 437.605,A -85,B 0,C 180,E1 -22037.341,E2 -22037.341} C_VEL
LIN {X 0,Y 183.922,Z 442.733,A -85,B 0,C 180,E1 -22040.098,E2 -22040.098} C_VEL
LIN {X 0,Y 183.811,Z 448.131,A -85,B 0,C 180,E1 -22043.781,E2 -22043.781} C_VEL
LIN {X 0,Y 183.797,Z 451.31,A -85,B 0,C 180,E1 -22046.711,E2 -22046.711} C_VEL
LIN {X 0,Y 184.178,Z 453.87,A -85,B 0,C 180,E1 -22049.999,E2 -22049.999} C_VEL
LIN {X 0,Y 183.525,Z 455.585,A -85,B 0,C 180,E1 -22054.392,E2 -22054.392} C_VEL
LIN {X 0,Y 183.458,Z 455.633,A -85,B 0,C 180,E1 -22058.814,E2 -22058.814} C_VEL
LIN {X 0,Y 184.353,Z 454.156,A -85,B 0,C 180,E1 -22063.222,E2 -22063.222} C_VEL
LIN {X 0,Y 185.255,Z 452.852,A -85,B 0,C 180,E1 -22065.4,E2 -22065.4} C_VEL
LIN {X 0,Y 187.216,Z 450.127,A -85,B 0,C 180,E1 -22068.607,E2 -22068.607} C_VEL
LIN {X 0,Y 189.746,Z 446.444,A -85,B 0,C 180,E1 -22071.739,E2 -22071.739} C_VEL
LIN {X 0,Y 192.777,Z 441.736,A -85,B 0,C 180,E1 -22074.787,E2 -22074.787} C_VEL
LIN {X 0,Y 197.299,Z 434.822,A -85,B 0,C 180,E1 -22078.162,E2 -22078.162} C_VEL
LIN {X 0,Y 201.827,Z 427.422,A -85,B 0,C 180,E1 -22080.905,E2 -22080.905} C_VEL
LIN {X 0,Y 206.84,Z 418.376,A -85,B 0,C 180,E1 -22083.514,E2 -22083.514} C_VEL
LIN {X 0,Y 211.463,Z 409.209,A -85,B 0,C 180,E1 -22085.564,E2 -22085.564} C_VEL
LIN {X 0,Y 216.463,Z 397.995,A -85,B 0,C 180,E1 -22087.5,E2 -22087.5} C_VEL
LIN {X 0,Y 220.76,Z 386.95,A -85,B 0,C 180,E1 -22088.957,E2 -22088.957} C_VEL
LIN {X 0,Y 224.753,Z 374.794,A -85,B 0,C 180,E1 -22090.161,E2 -22090.161} C_VEL
LIN {X 0,Y 228.066,Z 361.394,A -85,B 0,C 180,E1 -22091.151,E2 -22091.151} C_VEL
LIN {X 0,Y 230.462,Z 347.671,A -85,B 0,C 180,E1 -22091.869,E2 -22091.869} C_VEL
LIN {X 0,Y 233.568,Z 317.845,A -85,B 0,C 180,E1 -22092.986,E2 -22092.986} C_VEL
LIN {X 0,Y 233.409,Z 304.813,A -85,B 0,C 180,E1 -22094.105,E2 -22094.105} C_VEL
LIN {X 0,Y 231.878,Z 299.82,A -85,B 0,C 180,E1 -22095.216,E2 -22095.216} C_VEL
LIN {X 0,Y 229.437,Z 293.531,A -85,B 0,C 180,E1 -22096.965,E2 -22096.965} C_VEL
LIN {X 0,Y 226.957,Z 287.621,A -85,B 0,C 180,E1 -22098.98,E2 -22098.98} C_VEL
LIN {X 0,Y 223.696,Z 280.28,A -85,B 0,C 180,E1 -22102.112,E2 -22102.112} C_VEL
LIN {X 0,Y 220.896,Z 274.446,A -85,B 0,C 180,E1 -22105.647,E2 -22105.647} C_VEL
LIN {X 0,Y 218.519,Z 269.673,A -85,B 0,C 180,E1 -22110.628,E2 -22110.628} C_VEL
LIN {X 0,Y 217.995,Z 268.104,A -85,B 0,C 180,E1 -22114.514,E2 -22114.514} C_VEL
LIN {X 0,Y 218.535,Z 267.944,A -85,B 0,C 180,E1 -22117.9,E2 -22117.9} C_VEL
LIN {X 0,Y 219.834,Z 268.839,A -85,B 0,C 180,E1 -22120.999,E2 -22120.999} C_VEL
LIN {X 0,Y 221.75,Z 271.829,A -85,B 0,C 180,E1 -22124.12,E2 -22124.12} C_VEL
LIN {X 0,Y 222.696,Z 272.895,A -85,B 0,C 180,E1 -22125.278,E2 -22125.278} C_VEL
LIN {X 0,Y 225.771,Z 277.544,A -85,B 0,C 180,E1 -22128.401,E2 -22128.401} C_VEL
LIN {X 0,Y 228.419,Z 282.002,A -85,B 0,C 180,E1 -22130.606,E2 -22130.606} C_VEL
LIN {X 0,Y 231.674,Z 287.179,A -85,B 0,C 180,E1 -22132.896,E2 -22132.896} C_VEL
LIN {X 0,Y 235.476,Z 295.216,A -85,B 0,C 180,E1 -22135.318,E2 -22135.318} C_VEL
LIN {X 0,Y 235.404,Z 296.944,A -85,B 0,C 180,E1 -22135.43,E2 -22135.43} C_VEL
LIN {X 0,Y 231.489,Z 333.309,A -85,B 0,C 180,E1 -22136.845,E2 -22136.845} C_VEL
LIN {X 0,Y 229.602,Z 344.974,A -85,B 0,C 180,E1 -22137.588,E2 -22137.588} C_VEL
LIN {X 0,Y 226.649,Z 358.206,A -85,B 0,C 180,E1 -22138.77,E2 -22138.77} C_VEL
LIN {X 0,Y 223.177,Z 369.862,A -85,B 0,C 180,E1 -22140.152,E2 -22140.152} C_VEL
LIN {X 0,Y 219.058,Z 381.005,A -85,B 0,C 180,E1 -22141.838,E2 -22141.838} C_VEL
LIN {X 0,Y 214.843,Z 390.704,A -85,B 0,C 180,E1 -22143.751,E2 -22143.751} C_VEL
LIN {X 0,Y 209.814,Z 400.651,A -85,B 0,C 180,E1 -22146.25,E2 -22146.25} C_VEL
LIN {X 0,Y 204.949,Z 409.037,A -85,B 0,C 180,E1 -22149.017,E2 -22149.017} C_VEL
LIN {X 0,Y 200.145,Z 416.22,A -85,B 0,C 180,E1 -22152.163,E2 -22152.163} C_VEL
LIN {X 0,Y 195.531,Z 422.237,A -85,B 0,C 180,E1 -22155.793,E2 -22155.793} C_VEL
LIN {X 0,Y 192.039,Z 426.22,A -85,B 0,C 180,E1 -22159.23,E2 -22159.23} C_VEL
LIN {X 0,Y 189.616,Z 428.51,A -85,B 0,C 180,E1 -22162.089,E2 -22162.089} C_VEL
LIN {X 0,Y 187.209,Z 430.215,A -85,B 0,C 180,E1 -22165.714,E2 -22165.714} C_VEL
LIN {X 0,Y 185.386,Z 430.743,A -85,B 0,C 180,E1 -22169.527,E2 -22169.527} C_VEL
LIN {X 0,Y 184.283,Z 430.167,A -85,B 0,C 180,E1 -22172.965,E2 -22172.965} C_VEL
LIN {X 0,Y 183.638,Z 428.534,A -85,B 0,C 180,E1 -22176.517,E2 -22176.517} C_VEL
LIN {X 0,Y 183.516,Z 425.32,A -85,B 0,C 180,E1 -22180.62,E2 -22180.62} C_VEL
LIN {X 0,Y 183.86,Z 422.124,A -85,B 0,C 180,E1 -22183.476,E2 -22183.476} C_VEL
LIN {X 0,Y 184.643,Z 416.628,A -85,B 0,C 180,E1 -22187.253,E2 -22187.253} C_VEL
LIN {X 0,Y 185.572,Z 410.729,A -85,B 0,C 180,E1 -22190.391,E2 -22190.391} C_VEL
LIN {X 0,Y 186.945,Z 403.181,A -85,B 0,C 180,E1 -22193.601,E2 -22193.601} C_VEL
LIN {X 0,Y 188.669,Z 394.375,A -85,B 0,C 180,E1 -22196.604,E2 -22196.604} C_VEL
LIN {X 0,Y 190.366,Z 385.009,A -85,B 0,C 180,E1 -22199.174,E2 -22199.174} C_VEL
LIN {X 0,Y 192.364,Z 373.656,A -85,B 0,C 180,E1 -22201.644,E2 -22201.644} C_VEL
LIN {X 0,Y 194.183,Z 361.776,A -85,B 0,C 180,E1 -22203.682,E2 -22203.682} C_VEL
LIN {X 0,Y 195.857,Z 348.973,A -85,B 0,C 180,E1 -22205.346,E2 -22205.346} C_VEL
LIN {X 0,Y 197.192,Z 335.399,A -85,B 0,C 180,E1 -22206.641,E2 -22206.641} C_VEL
LIN {X 0,Y 198.031,Z 322.507,A -85,B 0,C 180,E1 -22207.462,E2 -22207.462} C_VEL
LIN {X 0,Y 200.858,Z 268.297,A -85,B 0,C 180,E1 -22209.787,E2 -22209.787} C_VEL
LIN {X 0,Y 191.031,Z 244.107,A -85,B 0,C 180,E1 -22212.193,E2 -22212.193} C_VEL
LIN {X 0,Y 185.834,Z 232.092,A -85,B 0,C 180,E1 -22213.523,E2 -22213.523} C_VEL
LIN {X 0,Y 185.704,Z 231.353,A -85,B 0,C 180,E1 -22213.652,E2 -22213.652} C_VEL
LIN {X 0,Y 185.894,Z 231.33,A -85,B 0,C 180,E1 -22219.41,E2 -22219.41} C_VEL
LIN {X 0,Y 185.937,Z 231.323,A -85,B 0,C 180,E1 -22223.49,E2 -22223.49} C_VEL
LIN {X 0,Y 186.203,Z 231.289,A -85,B 0,C 180,E1 -22227.838,E2 -22227.838} C_VEL
LIN {X 0,Y 186.402,Z 231.265,A -85,B 0,C 180,E1 -22230.001,E2 -22230.001} C_VEL
LIN {X 0,Y 185.905,Z 231.328,A -85,B 0,C 180,E1 -22234.337,E2 -22234.337} C_VEL
LIN {X 0,Y 185.98,Z 231.317,A -85,B 0,C 180,E1 -22238.695,E2 -22238.695} C_VEL
LIN {X 0,Y 185.731,Z 231.348,A -85,B 0,C 180,E1 -22243.123,E2 -22243.123} C_VEL
LIN {X 0,Y 185.692,Z 231.353,A -85,B 0,C 180,E1 -22247.625,E2 -22247.625} C_VEL
LIN {X 0,Y 185.579,Z 231.353,A -85,B 0,C 180,E1 -22252.254,E2 -22252.254} C_VEL
LIN {X 0,Y 185.51,Z 231.375,A -85,B 0,C 180,E1 -22257.041,E2 -22257.041} C_VEL
LIN {X 0,Y 185.545,Z 231.373,A -85,B 0,C 180,E1 -22259.5,E2 -22259.5} C_VEL
LIN {X 0,Y 185.498,Z 231.365,A -85,B 0,C 180,E1 -22264.633,E2 -22264.633} C_VEL
LIN {X 0,Y 185.501,Z 231.351,A -85,B 0,C 180,E1 -22267.315,E2 -22267.315} C_VEL
LIN {X 0,Y 185.465,Z 231.365,A -85,B 0,C 180,E1 -22270.722,E2 -22270.722} C_VEL
LIN {X 0,Y 185.459,Z 231.382,A -85,B 0,C 180,E1 -22276.056,E2 -22276.056} C_VEL
LIN {X 0,Y 185.461,Z 231.38,A -85,B 0,C 180,E1 -22279.893,E2 -22279.893} C_VEL
LIN {X 0,Y 185.504,Z 231.37,A -85,B 0,C 180,E1 -22282.714,E2 -22282.714} C_VEL
LIN {X 0,Y 185.533,Z 231.373,A -85,B 0,C 180,E1 -22287.973,E2 -22287.973} C_VEL
LIN {X 0,Y 185.549,Z 231.371,A -85,B 0,C 180,E1 -22290.596,E2 -22290.596} C_VEL
LIN {X 0,Y 185.583,Z 231.362,A -85,B 0,C 180,E1 -22295.382,E2 -22295.382} C_VEL
LIN {X 0,Y 185.675,Z 231.355,A -85,B 0,C 180,E1 -22301.136,E2 -22301.136} C_VEL
LIN {X 0,Y 185.685,Z 231.347,A -85,B 0,C 180,E1 -22304.637,E2 -22304.637} C_VEL
LIN {X 0,Y 185.891,Z 231.299,A -85,B 0,C 180,E1 -22309.419,E2 -22309.419} C_VEL
LIN {X 0,Y 185.936,Z 231.308,A -85,B 0,C 180,E1 -22313.489,E2 -22313.489} C_VEL
LIN {X 0,Y 186.2,Z 231.288,A -85,B 0,C 180,E1 -22317.837,E2 -22317.837} C_VEL
LIN {X 0,Y 186.384,Z 231.268,A -85,B 0,C 180,E1 -22320,E2 -22320} C_VEL
LIN {X 0,Y 185.89,Z 231.322,A -85,B 0,C 180,E1 -22324.337,E2 -22324.337} C_VEL
LIN {X 0,Y 185.979,Z 231.301,A -85,B 0,C 180,E1 -22328.694,E2 -22328.694} C_VEL
LIN {X 0,Y 185.719,Z 231.349,A -85,B 0,C 180,E1 -22333.124,E2 -22333.124} C_VEL
LIN {X 0,Y 185.658,Z 231.36,A -85,B 0,C 180,E1 -22337.628,E2 -22337.628} C_VEL
LIN {X 0,Y 185.556,Z 231.365,A -85,B 0,C 180,E1 -22342.257,E2 -22342.257} C_VEL
LIN {X 0,Y 185.504,Z 231.38,A -85,B 0,C 180,E1 -22347.041,E2 -22347.041} C_VEL
LIN {X 0,Y 185.546,Z 231.369,A -85,B 0,C 180,E1 -22349.499,E2 -22349.499} C_VEL
LIN {X 0,Y 185.499,Z 231.377,A -85,B 0,C 180,E1 -22354.632,E2 -22354.632} C_VEL
LIN {X 0,Y 185.502,Z 231.379,A -85,B 0,C 180,E1 -22357.314,E2 -22357.314} C_VEL
LIN {X 0,Y 185.464,Z 231.385,A -85,B 0,C 180,E1 -22360.721,E2 -22360.721} C_VEL
LIN {X 0,Y 185.457,Z 231.383,A -85,B 0,C 180,E1 -22366.056,E2 -22366.056} C_VEL
LIN {X 0,Y 185.519,Z 231.515,A -85,B 0,C 180,E1 -22368.161,E2 -22368.161} C_VEL
LIN {X 0,Y 187.733,Z 241.138,A -85,B 0,C 180,E1 -22372.607,E2 -22372.607} C_VEL
LIN {X 0,Y 188.429,Z 244.483,A -85,B 0,C 180,E1 -22374.065,E2 -22374.065} C_VEL
LIN {X 0,Y 195.387,Z 265.186,A -85,B 0,C 180,E1 -22376.013,E2 -22376.013} C_VEL
LIN {X 0,Y 199.342,Z 311.479,A -85,B 0,C 180,E1 -22378.733,E2 -22378.733} C_VEL
LIN {X 0,Y 197.155,Z 352.854,A -85,B 0,C 180,E1 -22380.546,E2 -22380.546} C_VEL
LIN {X 0,Y 196.168,Z 358.6,A -85,B 0,C 180,E1 -22380.822,E2 -22380.822} C_VEL
LIN {X 0,Y 192.561,Z 367.709,A -85,B 0,C 180,E1 -22381.287,E2 -22381.287} C_VEL
LIN {X 0,Y 188.633,Z 376.58,A -85,B 0,C 180,E1 -22381.972,E2 -22381.972} C_VEL
LIN {X 0,Y 187.163,Z 381.965,A -85,B 0,C 180,E1 -22382.59,E2 -22382.59} C_VEL
LIN {X 0,Y 185.151,Z 394.051,A -85,B 0,C 180,E1 -22384.419,E2 -22384.419} C_VEL
LIN {X 0,Y 183.135,Z 404.867,A -85,B 0,C 180,E1 -22386.537,E2 -22386.537} C_VEL
LIN {X 0,Y 181.137,Z 414.989,A -85,B 0,C 180,E1 -22389.049,E2 -22389.049} C_VEL
LIN {X 0,Y 179.448,Z 423.704,A -85,B 0,C 180,E1 -22391.74,E2 -22391.74} C_VEL
LIN {X 0,Y 178.209,Z 431.138,A -85,B 0,C 180,E1 -22394.561,E2 -22394.561} C_VEL
LIN {X 0,Y 177.148,Z 438.389,A -85,B 0,C 180,E1 -22397.978,E2 -22397.978} C_VEL
LIN {X 0,Y 176.77,Z 443.269,A -85,B 0,C 180,E1 -22400.849,E2 -22400.849} C_VEL
LIN {X 0,Y 176.76,Z 447.227,A -85,B 0,C 180,E1 -22403.725,E2 -22403.725} C_VEL
LIN {X 0,Y 176.747,Z 450.314,A -85,B 0,C 180,E1 -22406.58,E2 -22406.58} C_VEL
